LIN {X 0,Y 195.738,Z 380.154,A -85,B 0,C 180,E1 -22076.15,E2 -22076.15} C_VEL
LIN {X 0,Y 199.662,Z 372.613,A -85,B 0,C 180,E1 -22078.944,E2 -22078.944} C_VEL
LIN {X 0,Y 204.162,Z 363.072,A -85,B 0,C 180,E1 -22081.663,E2 -22081.663} C_VEL
LIN {X 0,Y 208.26,Z 353.291,A -85,B 0,C 180,E1 -22083.833,E2 -22083.833} C_VEL
LIN {X 0,Y 212.222,Z 342.404,A -85,B 0,C 180,E1 -22085.706,E2 -22085.706} C_VEL
LIN {X 0,Y 216.03,Z 330.178,A -85,B 0,C 180,E1 -22087.292,E2 -22087.292} C_VEL
LIN {X 0,Y 218.974,Z 318.329,A -85,B 0,C 180,E1 -22088.448,E2 -22088.448} C_VEL
LIN {X 0,Y 221.492,Z 304.57,A -85,B 0,C 180,E1 -22089.388,E2 -22089.388} C_VEL
LIN {X 0,Y 223.101,Z 291.496,A -85,B 0,C 180,E1 -22089.946,E2 -22089.946} C_VEL
LIN {X 0,Y 226.073,Z 252.422,A -85,B 0,C 180,E1 -22091.263,E2 -22091.263} C_VEL
LIN {X 0,Y 221.932,Z 242.001,A -85,B 0,C 180,E1 -22093.251,E2 -22093.251} C_VEL
LIN {X 0,Y 217.229,Z 232.155,A -85,B 0,C 180,E1 -22095.657,E2 -22095.657} C_VEL
LIN {X 0,Y 212.28,Z 223.234,A -85,B 0,C 180,E1 -22098.469,E2 -22098.469} C_VEL
LIN {X 0,Y 208.755,Z 217.596,A -85,B 0,C 180,E1 -22100.701,E2 -22100.701} C_VEL
LIN {X 0,Y 205.495,Z 212.523,A -85,B 0,C 180,E1 -22103.083,E2 -22103.083} C_VEL
LIN {X 0,Y 201.551,Z 206.784,A -85,B 0,C 180,E1 -22106.493,E2 -22106.493} C_VEL
LIN {X 0,Y 198.426,Z 202.606,A -85,B 0,C 180,E1 -22109.907,E2 -22109.907} C_VEL
LIN {X 0,Y 196.823,Z 200.527,A -85,B 0,C 180,E1 -22112.153,E2 -22112.153} C_VEL
LIN {X 0,Y 194.604,Z 197.984,A -85,B 0,C 180,E1 -22116.592,E2 -22116.592} C_VEL
LIN {X 0,Y 193.638,Z 197.163,A -85,B 0,C 180,E1 -22120.933,E2 -22120.933} C_VEL
LIN {X 0,Y 194.019,Z 197.379,A -85,B 0,C 180,E1 -22125.724,E2 -22125.724} C_VEL
LIN {X 0,Y 196.637,Z 198.991,A -85,B 0,C 180,E1 -22131.58,E2 -22131.58} C_VEL
LIN {X 0,Y 197.623,Z 200.557,A -85,B 0,C 180,E1 -22133.135,E2 -22133.135} C_VEL
LIN {X 0,Y 199.349,Z 203.037,A -85,B 0,C 180,E1 -22135.386,E2 -22135.386} C_VEL
LIN {X 0,Y 201.956,Z 205.11,A -85,B 0,C 180,E1 -22137.911,E2 -22137.911} C_VEL
LIN {X 0,Y 206.643,Z 212.032,A -85,B 0,C 180,E1 -22141.857,E2 -22141.857} C_VEL
LIN {X 0,Y 209.872,Z 216.687,A -85,B 0,C 180,E1 -22144.105,E2 -22144.105} C_VEL
LIN {X 0,Y 213.368,Z 222.386,A -85,B 0,C 180,E1 -22146.258,E2 -22146.258} C_VEL
LIN {X 0,Y 218.333,Z 231.127,A -85,B 0,C 180,E1 -22148.992,E2 -22148.992} C_VEL
LIN {X 0,Y 223.137,Z 241.11,A -85,B 0,C 180,E1 -22151.401,E2 -22151.401} C_VEL
LIN {X 0,Y 226.339,Z 248.713,A -85,B 0,C 180,E1 -22152.893,E2 -22152.893} C_VEL
LIN {X 0,Y 222.66,Z 293.735,A -85,B 0,C 180,E1 -22154.419,E2 -22154.419} C_VEL
LIN {X 0,Y 220.636,Z 307.167,A -85,B 0,C 180,E1 -22155.172,E2 -22155.172} C_VEL
LIN {X 0,Y 218.273,Z 318.852,A -85,B 0,C 180,E1 -22156.154,E2 -22156.154} C_VEL
LIN {X 0,Y 215.211,Z 330.433,A -85,B 0,C 180,E1 -22157.458,E2 -22157.458} C_VEL
LIN {X 0,Y 211.4,Z 342.253,A -85,B 0,C 180,E1 -22159.22,E2 -22159.22} C_VEL
LIN {X 0,Y 207.441,Z 352.476,A -85,B 0,C 180,E1 -22161.161,E2 -22161.161} C_VEL
LIN {X 0,Y 203.182,Z 362.202,A -85,B 0,C 180,E1 -22163.57,E2 -22163.57} C_VEL
LIN {X 0,Y 199.338,Z 369.905,A -85,B 0,C 180,E1 -22165.974,E2 -22165.974} C_VEL
LIN {X 0,Y 195.765,Z 376.759,A -85,B 0,C 180,E1 -22168.717,E2 -22168.717} C_VEL
LIN {X 0,Y 192.541,Z 382.26,A -85,B 0,C 180,E1 -22171.489,E2 -22171.489} C_VEL
LIN {X 0,Y 189.175,Z 387.791,A -85,B 0,C 180,E1 -22175.188,E2 -22175.188} C_VEL
LIN {X 0,Y 187.173,Z 390.817,A -85,B 0,C 180,E1 -22177.958,E2 -22177.958} C_VEL
LIN {X 0,Y 185.559,Z 393.091,A -85,B 0,C 180,E1 -22180.761,E2 -22180.761} C_VEL
LIN {X 0,Y 184.378,Z 394.674,A -85,B 0,C 180,E1 -22183.599,E2 -22183.599} C_VEL
LIN {X 0,Y 183.413,Z 395.581,A -85,B 0,C 180,E1 -22186.721,E2 -22186.721} C_VEL
LIN {X 0,Y 182.76,Z 395.654,A -85,B 0,C 180,E1 -22190.271,E2 -22190.271} C_VEL
LIN {X 0,Y 182.533,Z 394.645,A -85,B 0,C 180,E1 -22193.953,E2 -22193.953} C_VEL
LIN {X 0,Y 182.717,Z 392.379,A -85,B 0,C 180,E1 -22197.799,E2 -22197.799} C_VEL
LIN {X 0,Y 183.447,Z 388.592,A -85,B 0,C 180,E1 -22201.779,E2 -22201.779} C_VEL
LIN {X 0,Y 184.329,Z 384.06,A -85,B 0,C 180,E1 -22205.206,E2 -22205.206} C_VEL
LIN {X 0,Y 185.721,Z 377.57,A -85,B 0,C 180,E1 -22208.933,E2 -22208.933} C_VEL
LIN {X 0,Y 187.317,Z 370.754,A -85,B 0,C 180,E1 -22211.972,E2 -22211.972} C_VEL
LIN {X 0,Y 189.403,Z 362.35,A -85,B 0,C 180,E1 -22214.948,E2 -22214.948} C_VEL
LIN {X 0,Y 191.822,Z 352.236,A -85,B 0,C 180,E1 -22217.793,E2 -22217.793} C_VEL
LIN {X 0,Y 194.205,Z 341.694,A -85,B 0,C 180,E1 -22220.104,E2 -22220.104} C_VEL
LIN {X 0,Y 196.607,Z 329.365,A -85,B 0,C 180,E1 -22222.214,E2 -22222.214} C_VEL
LIN {X 0,Y 198.503,Z 317.646,A -85,B 0,C 180,E1 -22223.736,E2 -22223.736} C_VEL
LIN {X 0,Y 200.201,Z 303.923,A -85,B 0,C 180,E1 -22225.03,E2 -22225.03} C_VEL
LIN {X 0,Y 201.472,Z 291.153,A -85,B 0,C 180,E1 -22225.814,E2 -22225.814} C_VEL
LIN {X 0,Y 204.341,Z 231.553,A -85,B 0,C 180,E1 -22228.072,E2 -22228.072} C_VEL
LIN {X 0,Y 198.187,Z 214.042,A -85,B 0,C 180,E1 -22229.769,E2 -22229.769} C_VEL
LIN {X 0,Y 191.241,Z 196.738,A -85,B 0,C 180,E1 -22231.713,E2 -22231.713} C_VEL
LIN {X 0,Y 186.943,Z 189.387,A -85,B 0,C 180,E1 -22232.819,E2 -22232.819} C_VEL
LIN {X 0,Y 186.099,Z 187.307,A -85,B 0,C 180,E1 -22233.25,E2 -22233.25} C_VEL
LIN {X 0,Y 185.982,Z 186.84,A -85,B 0,C 180,E1 -22233.794,E2 -22233.794} C_VEL
LIN {X 0,Y 185.98,Z 186.809,A -85,B 0,C 180,E1 -22238.696,E2 -22238.696} C_VEL
LIN {X 0,Y 185.726,Z 186.836,A -85,B 0,C 180,E1 -22243.125,E2 -22243.125} C_VEL
LIN {X 0,Y 185.69,Z 186.842,A -85,B 0,C 180,E1 -22247.627,E2 -22247.627} C_VEL
LIN {X 0,Y 185.597,Z 186.866,A -85,B 0,C 180,E1 -22252.253,E2 -22252.253} C_VEL
LIN {X 0,Y 185.561,Z 186.846,A -85,B 0,C 180,E1 -22257.034,E2 -22257.034} C_VEL
LIN {X 0,Y 185.578,Z 186.864,A -85,B 0,C 180,E1 -22259.495,E2 -22259.495} C_VEL
LIN {X 0,Y 185.499,Z 186.853,A -85,B 0,C 180,E1 -22264.634,E2 -22264.634} C_VEL
LIN {X 0,Y 185.506,Z 186.847,A -85,B 0,C 180,E1 -22267.315,E2 -22267.315} C_VEL
LIN {X 0,Y 185.473,Z 186.879,A -85,B 0,C 180,E1 -22270.727,E2 -22270.727} C_VEL
LIN {X 0,Y 185.48,Z 186.875,A -85,B 0,C 180,E1 -22273.953,E2 -22273.953} C_VEL
LIN {X 0,Y 185.472,Z 186.839,A -85,B 0,C 180,E1 -22279.278,E2 -22279.278} C_VEL
LIN {X 0,Y 185.506,Z 186.867,A -85,B 0,C 180,E1 -22282.714,E2 -22282.714} C_VEL
LIN {X 0,Y 185.533,Z 186.866,A -85,B 0,C 180,E1 -22287.974,E2 -22287.974} C_VEL
LIN {X 0,Y 185.55,Z 186.865,A -85,B 0,C 180,E1 -22290.597,E2 -22290.597} C_VEL
LIN {X 0,Y 185.584,Z 186.862,A -85,B 0,C 180,E1 -22295.383,E2 -22295.383} C_VEL
LIN {X 0,Y 185.678,Z 186.854,A -85,B 0,C 180,E1 -22301.135,E2 -22301.135} C_VEL
LIN {X 0,Y 185.697,Z 186.839,A -85,B 0,C 180,E1 -22304.638,E2 -22304.638} C_VEL
LIN {X 0,Y 185.892,Z 186.827,A -85,B 0,C 180,E1 -22309.421,E2 -22309.421} C_VEL
LIN {X 0,Y 185.933,Z 186.815,A -85,B 0,C 180,E1 -22313.49,E2 -22313.49} C_VEL
LIN {X 0,Y 186.18,Z 186.789,A -85,B 0,C 180,E1 -22317.838,E2 -22317.838} C_VEL
LIN {X 0,Y 186.383,Z 186.749,A -85,B 0,C 180,E1 -22320.001,E2 -22320.001} C_VEL
LIN {X 0,Y 185.888,Z 186.787,A -85,B 0,C 180,E1 -22324.338,E2 -22324.338} C_VEL
LIN {X 0,Y 185.98,Z 186.816,A -85,B 0,C 180,E1 -22328.695,E2 -22328.695} C_VEL
LIN {X 0,Y 185.72,Z 186.835,A -85,B 0,C 180,E1 -22333.124,E2 -22333.124} C_VEL
LIN {X 0,Y 185.656,Z 186.834,A -85,B 0,C 180,E1 -22337.629,E2 -22337.629} C_VEL
LIN {X 0,Y 185.545,Z 186.871,A -85,B 0,C 180,E1 -22342.259,E2 -22342.259} C_VEL
LIN {X 0,Y 185.502,Z 186.856,A -85,B 0,C 180,E1 -22347.043,E2 -22347.043} C_VEL
LIN {X 0,Y 185.549,Z 186.872,A -85,B 0,C 180,E1 -22349.499,E2 -22349.499} C_VEL
LIN {X 0,Y 185.502,Z 186.86,A -85,B 0,C 180,E1 -22354.632,E2 -22354.632} C_VEL
LIN {X 0,Y 185.505,Z 186.878,A -85,B 0,C 180,E1 -22357.314,E2 -22357.314} C_VEL
LIN {X 0,Y 185.466,Z 186.869,A -85,B 0,C 180,E1 -22360.721,E2 -22360.721} C_VEL
LIN {X 0,Y 185.46,Z 186.875,A -85,B 0,C 180,E1 -22366.056,E2 -22366.056} C_VEL
LIN {X 0,Y 185.55,Z 187.033,A -85,B 0,C 180,E1 -22369.248,E2 -22369.248} C_VEL
LIN {X 0,Y 186.204,Z 189.727,A -85,B 0,C 180,E1 -22370.753,E2 -22370.753} C_VEL
LIN {X 0,Y 189.464,Z 197.093,A -85,B 0,C 180,E1 -22371.776,E2 -22371.776} C_VEL
LIN {X 0,Y 196.233,Z 213.271,A -85,B 0,C 180,E1 -22373.674,E2 -22373.674} C_VEL
LIN {X 0,Y 202.546,Z 230.72,A -85,B 0,C 180,E1 -22375.415,E2 -22375.415} C_VEL
LIN {X 0,Y 204.066,Z 243.654,A -85,B 0,C 180,E1 -22376.204,E2 -22376.204} C_VEL
LIN {X 0,Y 201.845,Z 288.233,A -85,B 0,C 180,E1 -22377.856,E2 -22377.856} C_VEL
LIN {X 0,Y 200.846,Z 294.037,A -85,B 0,C 180,E1 -22377.992,E2 -22377.992} C_VEL
LIN {X 0,Y 197.428,Z 303.347,A -85,B 0,C 180,E1 -22378.124,E2 -22378.124} C_VEL
LIN {X 0,Y 193.839,Z 312.517,A -85,B 0,C 180,E1 -22378.473,E2 -22378.473} C_VEL
LIN {X 0,Y 192.575,Z 318.098,A -85,B 0,C 180,E1 -22378.925,E2 -22378.925} C_VEL
LIN {X 0,Y 190.816,Z 329.003,A -85,B 0,C 180,E1 -22380.181,E2 -22380.181} C_VEL
LIN {X 0,Y 188.47,Z 340.49,A -85,B 0,C 180,E1 -22381.913,E2 -22381.913} C_VEL
LIN {X 0,Y 186.206,Z 351.023,A -85,B 0,C 180,E1 -22383.973,E2 -22383.973} C_VEL
LIN {X 0,Y 183.947,Z 360.69,A -85,B 0,C 180,E1 -22386.348,E2 -22386.348} C_VEL
LIN {X 0,Y 181.855,Z 369.512,A -85,B 0,C 180,E1 -22389.052,E2 -22389.052} C_VEL
LIN {X 0,Y 179.616,Z 378.019,A -85,B 0,C 180,E1 -22392.345,E2 -22392.345} C_VEL
LIN {X 0,Y 177.933,Z 384.849,A -85,B 0,C 180,E1 -22395.706,E2 -22395.706} C_VEL
LIN {X 0,Y 176.715,Z 391.092,A -85,B 0,C 180,E1 -22399.688,E2 -22399.688} C_VEL
LIN {X 0,Y 176.144,Z 395.11,A -85,B 0,C 180,E1 -22403.123,E2 -22403.123} C_VEL
LIN {X 0,Y 175.914,Z 398.454,A -85,B 0,C 180,E1 -22407.193,E2 -22407.193} C_VEL
LIN {X 0,Y 176.006,Z 399.99,A -85,B 0,C 180,E1 -22409.998,E2 -22409.998} C_VEL
LIN {X 0,Y 175.913,Z 400.846,A -85,B 0,C 180,E1 -22412.802,E2 -22412.802} C_VEL
LIN {X 0,Y 176.239,Z 401.057,A -85,B 0,C 180,E1 -22416.868,E2 -22416.868} C_VEL
LIN {X 0,Y 176.61,Z 400.64,A -85,B 0,C 180,E1 -22419.156,E2 -22419.156} C_VEL
LIN {X 0,Y 177.235,Z 399.821,A -85,B 0,C 180,E1 -22421.433,E2 -22421.433} C_VEL
LIN {X 0,Y 179.194,Z 396.958,A -85,B 0,C 180,E1 -22425.932,E2 -22425.932} C_VEL
LIN {X 0,Y 181.363,Z 393.721,A -85,B 0,C 180,E1 -22429.229,E2 -22429.229} C_VEL
LIN {X 0,Y 184.319,Z 389.441,A -85,B 0,C 180,E1 -22432.411,E2 -22432.411} C_VEL
LIN {X 0,Y 187.559,Z 384.03,A -85,B 0,C 180,E1 -22435.523,E2 -22435.523} C_VEL
LIN {X 0,Y 191.342,Z 377.304,A -85,B 0,C 180,E1 -22438.519,E2 -22438.519} C_VEL
LIN {X 0,Y 195.81,Z 369.003,A -85,B 0,C 180,E1 -22441.358,E2 -22441.358} C_VEL
LIN {X 0,Y 199.93,Z 360.528,A -85,B 0,C 180,E1 -22443.615,E2 -22443.615} C_VEL
LIN {X 0,Y 203.851,Z 351.332,A -85,B 0,C 180,E1 -22445.573,E2 -22445.573} C_VEL
LIN {X 0,Y 207.573,Z 341.406,A -85,B 0,C 180,E1 -22447.241,E2 -22447.241} C_VEL
LIN {X 0,Y 211.532,Z 328.981,A -85,B 0,C 180,E1 -22448.834,E2 -22448.834} C_VEL
LIN {X 0,Y 214.644,Z 316.652,A -85,B 0,C 180,E1 -22449.981,E2 -22449.981} C_VEL
LIN {X 0,Y 217.164,Z 302.775,A -85,B 0,C 180,E1 -22450.901,E2 -22450.901} C_VEL
LIN {X 0,Y 218.781,Z 288.708,A -85,B 0,C 180,E1 -22451.459,E2 -22451.459} C_VEL
LIN {X 0,Y 221.477,Z 254.949,A -85,B 0,C 180,E1 -22452.601,E2 -22452.601} C_VEL
LIN {X 0,Y 217.87,Z 245.778,A -85,B 0,C 180,E1 -22454.493,E2 -22454.493} C_VEL
LIN {X 0,Y 214.01,Z 237.383,A -85,B 0,C 180,E1 -22456.613,E2 -22456.613} C_VEL
LIN {X 0,Y 209.331,Z 228.687,A -85,B 0,C 180,E1 -22459.461,E2 -22459.461} C_VEL
LIN {X 0,Y 206.424,Z 223.698,A -85,B 0,C 180,E1 -22461.459,E2 -22461.459} C_VEL
LIN {X 0,Y 203.273,Z 218.661,A -85,B 0,C 180,E1 -22463.886,E2 -22463.886} C_VEL
LIN {X 0,Y 199.948,Z 213.504,A -85,B 0,C 180,E1 -22466.966,E2 -22466.966} C_VEL
LIN {X 0,Y 196.83,Z 209.093,A -85,B 0,C 180,E1 -22470.603,E2 -22470.603} C_VEL
LIN {X 0,Y 195.104,Z 206.982,A -85,B 0,C 180,E1 -22473.193,E2 -22473.193} C_VEL
LIN {X 0,Y 193.418,Z 204.91,A -85,B 0,C 180,E1 -22477.007,E2 -22477.007} C_VEL
LIN {X 0,Y 192.567,Z 204.165,A -85,B 0,C 180,E1 -22481.596,E2 -22481.596} C_VEL
LIN {X 0,Y 193.121,Z 204.542,A -85,B 0,C 180,E1 -22486.267,E2 -22486.267} C_VEL
LIN {X 0,Y 195.422,Z 205.908,A -85,B 0,C 180,E1 -22491.325,E2 -22491.325} C_VEL
LIN {X 0,Y 197.911,Z 209.845,A -85,B 0,C 180,E1 -22494.97,E2 -22494.97} C_VEL
LIN {X 0,Y 200.228,Z 211.717,A -85,B 0,C 180,E1 -22497.327,E2 -22497.327} C_VEL
LIN {X 0,Y 204.479,Z 218.281,A -85,B 0,C 180,E1 -22501.138,E2 -22501.138} C_VEL
LIN {X 0,Y 207.628,Z 223.06,A -85,B 0,C 180,E1 -22503.449,E2 -22503.449} C_VEL
LIN {X 0,Y 210.456,Z 227.855,A -85,B 0,C 180,E1 -22505.311,E2 -22505.311} C_VEL
LIN {X 0,Y 215.265,Z 236.702,A -85,B 0,C 180,E1 -22508.156,E2 -22508.156} C_VEL
LIN {X 0,Y 219.578,Z 246.025,A -85,B 0,C 180,E1 -22510.443,E2 -22510.443} C_VEL
LIN {X 0,Y 221.691,Z 251.168,A -85,B 0,C 180,E1 -22511.523,E2 -22511.523} C_VEL
LIN {X 0,Y 218.196,Z 293.227,A -85,B 0,C 180,E1 -22512.984,E2 -22512.984} C_VEL
LIN {X 0,Y 216.114,Z 306.637,A -85,B 0,C 180,E1 -22513.717,E2 -22513.717} C_VEL
LIN {X 0,Y 213.488,Z 319.191,A -85,B 0,C 180,E1 -22514.77,E2 -22514.77} C_VEL
LIN {X 0,Y 210.273,Z 330.755,A -85,B 0,C 180,E1 -22516.081,E2 -22516.081} C_VEL
LIN {X 0,Y 206.284,Z 342.543,A -85,B 0,C 180,E1 -22517.855,E2 -22517.855} C_VEL
LIN {X 0,Y 201.869,Z 353.33,A -85,B 0,C 180,E1 -22519.958,E2 -22519.958} C_VEL
LIN {X 0,Y 197.539,Z 362.643,A -85,B 0,C 180,E1 -22522.336,E2 -22522.336} C_VEL
LIN {X 0,Y 192.94,Z 371.273,A -85,B 0,C 180,E1 -22525.145,E2 -22525.145} C_VEL
LIN {X 0,Y 188.764,Z 378.65,A -85,B 0,C 180,E1 -22528.332,E2 -22528.332} C_VEL
LIN {X 0,Y 185.469,Z 383.845,A -85,B 0,C 180,E1 -22531.218,E2 -22531.218} C_VEL
LIN {X 0,Y 182.719,Z 388.005,A -85,B 0,C 180,E1 -22534.213,E2 -22534.213} C_VEL
LIN {X 0,Y 179.62,Z 392.216,A -85,B 0,C 180,E1 -22538.511,E2 -22538.511} C_VEL
LIN {X 0,Y 177.739,Z 394.503,A -85,B 0,C 180,E1 -22542.236,E2 -22542.236} C_VEL
LIN {X 0,Y 176.535,Z 395.633,A -85,B 0,C 180,E1 -22545.773,E2 -22545.773} C_VEL
LIN {X 0,Y 175.669,Z 395.73,A -85,B 0,C 180,E1 -22550.204,E2 -22550.204} C_VEL
LIN {X 0,Y 175.449,Z 394.899,A -85,B 0,C 180,E1 -22553.238,E2 -22553.238} C_VEL
LIN {X 0,Y 175.558,Z 392.775,A -85,B 0,C 180,E1 -22557.21,E2 -22557.21} C_VEL
LIN {X 0,Y 176.232,Z 389.094,A -85,B 0,C 180,E1 -22561.412,E2 -22561.412} C_VEL
LIN {X 0,Y 177.134,Z 384.659,A -85,B 0,C 180,E1 -22564.99,E2 -22564.99} C_VEL
LIN {X 0,Y 178.39,Z 378.734,A -85,B 0,C 180,E1 -22568.631,E2 -22568.631} C_VEL
LIN {X 0,Y 180.023,Z 372.156,A -85,B 0,C 180,E1 -22571.804,E2 -22571.804} C_VEL
LIN {X 0,Y 182.012,Z 364.235,A -85,B 0,C 180,E1 -22574.862,E2 -22574.862} C_VEL
LIN {X 0,Y 184.298,Z 355.24,A -85,B 0,C 180,E1 -22577.616,E2 -22577.616} C_VEL
LIN {X 0,Y 186.906,Z 344.31,A -85,B 0,C 180,E1 -22580.261,E2 -22580.261} C_VEL
LIN {X 0,Y 189.124,Z 333.821,A -85,B 0,C 180,E1 -22582.261,E2 -22582.261} C_VEL
LIN {X 0,Y 191.357,Z 321.68,A -85,B 0,C 180,E1 -22584.037,E2 -22584.037} C_VEL
LIN {X 0,Y 193.148,Z 308.919,A -85,B 0,C 180,E1 -22585.437,E2 -22585.437} C_VEL
LIN {X 0,Y 194.587,Z 295.907,A -85,B 0,C 180,E1 -22586.411,E2 -22586.411} C_VEL
LIN {X 0,Y 195.581,Z 280.594,A -85,B 0,C 180,E1 -22587.106,E2 -22587.106} C_VEL
LIN {X 0,Y 197.962,Z 233.103,A -85,B 0,C 180,E1 -22588.929,E2 -22588.929} C_VEL
LIN {X 0,Y 192.389,Z 217.271,A -85,B 0,C 180,E1 -22590.53,E2 -22590.53} C_VEL
LIN {X 0,Y 185.66,Z 200.398,A -85,B 0,C 180,E1 -22592.499,E2 -22592.499} C_VEL
LIN {X 0,Y 180.108,Z 190.85,A -85,B 0,C 180,E1 -22594.022,E2 -22594.022} C_VEL
LIN {X 0,Y 178.972,Z 188.334,A -85,B 0,C 180,E1 -22594.507,E2 -22594.507} C_VEL
LIN {X 0,Y 178.871,Z 187.736,A -85,B 0,C 180,E1 -22595.074,E2 -22595.074} C_VEL
LIN {X 0,Y 178.909,Z 187.691,A -85,B 0,C 180,E1 -22599.043,E2 -22599.043} C_VEL
LIN {X 0,Y 178.655,Z 187.718,A -85,B 0,C 180,E1 -22603.655,E2 -22603.655} C_VEL
LIN {X 0,Y 178.623,Z 187.716,A -85,B 0,C 180,E1 -22609.218,E2 -22609.218} C_VEL
LIN {X 0,Y 178.525,Z 187.727,A -85,B 0,C 180,E1 -22615.119,E2 -22615.119} C_VEL
LIN {X 0,Y 178.522,Z 187.747,A -85,B 0,C 180,E1 -22619.995,E2 -22619.995} C_VEL
LIN {X 0,Y 178.485,Z 187.729,A -85,B 0,C 180,E1 -22624.221,E2 -22624.221} C_VEL
LIN {X 0,Y 178.397,Z 187.749,A -85,B 0,C 180,E1 -22629.076,E2 -22629.076} C_VEL
LIN {X 0,Y 178.4,Z 187.762,A -85,B 0,C 180,E1 -22632.047,E2 -22632.047} C_VEL
LIN {X 0,Y 178.401,Z 187.746,A -85,B 0,C 180,E1 -22635.164,E2 -22635.164} C_VEL
LIN {X 0,Y 178.405,Z 187.715,A -85,B 0,C 180,E1 -22638.461,E2 -22638.461} C_VEL
LIN {X 0,Y 178.423,Z 187.756,A -85,B 0,C 180,E1 -22643.784,E2 -22643.784} C_VEL
LIN {X 0,Y 178.486,Z 187.75,A -85,B 0,C 180,E1 -22646.548,E2 -22646.548} C_VEL
LIN {X 0,Y 178.447,Z 187.755,A -85,B 0,C 180,E1 -22651.797,E2 -22651.797} C_VEL
LIN {X 0,Y 178.519,Z 187.742,A -85,B 0,C 180,E1 -22654.891,E2 -22654.891} C_VEL
LIN {X 0,Y 178.626,Z 187.733,A -85,B 0,C 180,E1 -22660.787,E2 -22660.787} C_VEL
LIN {X 0,Y 178.66,Z 187.722,A -85,B 0,C 180,E1 -22666.349,E2 -22666.349} C_VEL
LIN {X 0,Y 178.908,Z 187.691,A -85,B 0,C 180,E1 -22670.961,E2 -22670.961} C_VEL
LIN {X 0,Y 179.128,Z 187.668,A -85,B 0,C 180,E1 -22677.752,E2 -22677.752} C_VEL
LIN {X 0,Y 179.349,Z 187.625,A -85,B 0,C 180,E1 -22680.001,E2 -22680.001} C_VEL
LIN {X 0,Y 178.837,Z 187.665,A -85,B 0,C 180,E1 -22684.509,E2 -22684.509} C_VEL
LIN {X 0,Y 178.911,Z 187.697,A -85,B 0,C 180,E1 -22689.041,E2 -22689.041} C_VEL
LIN {X 0,Y 178.646,Z 187.711,A -85,B 0,C 180,E1 -22693.654,E2 -22693.654} C_VEL
LIN {X 0,Y 178.56,Z 187.733,A -85,B 0,C 180,E1 -22699.152,E2 -22699.152} C_VEL
LIN {X 0,Y 178.47,Z 187.728,A -85,B 0,C 180,E1 -22705.076,E2 -22705.076} C_VEL
LIN {X 0,Y 178.466,Z 187.755,A -85,B 0,C 180,E1 -22710.794,E2 -22710.794} C_VEL
LIN {X 0,Y 178.488,Z 187.731,A -85,B 0,C 180,E1 -22714.218,E2 -22714.218} C_VEL
LIN {X 0,Y 178.392,Z 187.751,A -85,B 0,C 180,E1 -22719.077,E2 -22719.077} C_VEL
LIN {X 0,Y 178.399,Z 187.76,A -85,B 0,C 180,E1 -22722.046,E2 -22722.046} C_VEL
LIN {X 0,Y 178.396,Z 187.751,A -85,B 0,C 180,E1 -22725.165,E2 -22725.165} C_VEL
LIN {X 0,Y 178.478,Z 187.975,A -85,B 0,C 180,E1 -22728.433,E2 -22728.433} C_VEL
LIN {X 0,Y 178.981,Z 189.888,A -85,B 0,C 180,E1 -22729.427,E2 -22729.427} C_VEL
LIN {X 0,Y 185.903,Z 205.264,A -85,B 0,C 180,E1 -22731.562,E2 -22731.562} C_VEL
LIN {X 0,Y 193.14,Z 223.627,A -85,B 0,C 180,E1 -22733.671,E2 -22733.671} C_VEL
LIN {X 0,Y 196.383,Z 232.984,A -85,B 0,C 180,E1 -22734.608,E2 -22734.608} C_VEL
LIN {X 0,Y 197.716,Z 244.563,A -85,B 0,C 180,E1 -22735.336,E2 -22735.336} C_VEL
LIN {X 0,Y 194.76,Z 298.7,A -85,B 0,C 180,E1 -22737.457,E2 -22737.457} C_VEL
LIN {X 0,Y 193.243,Z 312.548,A -85,B 0,C 180,E1 -22738.401,E2 -22738.401} C_VEL
LIN {X 0,Y 192.575,Z 318.098,A -85,B 0,C 180,E1 -22738.925,E2 -22738.925} C_VEL
LIN {X 0,Y 191.129,Z 323.594,A -85,B 0,C 180,E1 -22739.419,E2 -22739.419} C_VEL
LIN {X 0,Y 186.873,Z 332.206,A -85,B 0,C 180,E1 -22740.197,E2 -22740.197} C_VEL
LIN {X 0,Y 182.461,Z 340.458,A -85,B 0,C 180,E1 -22741.228,E2 -22741.228} C_VEL
LIN {X 0,Y 180.794,Z 345.385,A -85,B 0,C 180,E1 -22742.112,E2 -22742.112} C_VEL
LIN {X 0,Y 178.494,Z 355.276,A -85,B 0,C 180,E1 -22744.333,E2 -22744.333} C_VEL
LIN {X 0,Y 175.841,Z 365.552,A -85,B 0,C 180,E1 -22747.236,E2 -22747.236} C_VEL
LIN {X 0,Y 173.864,Z 373.06,A -85,B 0,C 180,E1 -22749.902,E2 -22749.902} C_VEL
LIN {X 0,Y 171.82,Z 380.848,A -85,B 0,C 180,E1 -22753.36,E2 -22753.36} C_VEL
LIN {X 0,Y 170.385,Z 387.089,A -85,B 0,C 180,E1 -22756.885,E2 -22756.885} C_VEL
LIN {X 0,Y 169.459,Z 392.013,A -85,B 0,C 180,E1 -22760.449,E2 -22760.449} C_VEL
LIN {X 0,Y 168.968,Z 395.766,A -85,B 0,C 180,E1 -22764.029,E2 -22764.029} C_VEL
LIN {X 0,Y 168.822,Z 398.459,A -85,B 0,C 180,E1 -22767.612,E2 -22767.612} C_VEL
LIN {X 0,Y 168.918,Z 399.716,A -85,B 0,C 180,E1 -22769.998,E2 -22769.998} C_VEL
LIN {X 0,Y 168.836,Z 400.584,A -85,B 0,C 180,E1 -22772.504,E2 -22772.504} C_VEL
LIN {X 0,Y 168.939,Z 400.957,A -85,B 0,C 180,E1 -22774.77,E2 -22774.77} C_VEL
LIN {X 0,Y 169.579,Z 400.602,A -85,B 0,C 180,E1 -22779.54,E2 -22779.54} C_VEL
LIN {X 0,Y 170.275,Z 399.859,A -85,B 0,C 180,E1 -22781.907,E2 -22781.907} C_VEL
LIN {X 0,Y 171.185,Z 398.703,A -85,B 0,C 180,E1 -22784.258,E2 -22784.258} C_VEL
LIN {X 0,Y 173.781,Z 395.152,A -85,B 0,C 180,E1 -22788.874,E2 -22788.874} C_VEL
LIN {X 0,Y 176.673,Z 391.337,A -85,B 0,C 180,E1 -22792.201,E2 -22792.201} C_VEL
LIN {X 0,Y 180.088,Z 386.439,A -85,B 0,C 180,E1 -22795.419,E2 -22795.419} C_VEL
LIN {X 0,Y 183.647,Z 380.584,A -85,B 0,C 180,E1 -22798.451,E2 -22798.451} C_VEL
LIN {X 0,Y 188.236,Z 372.834,A -85,B 0,C 180,E1 -22801.511,E2 -22801.511} C_VEL
LIN {X 0,Y 192.349,Z 365.182,A -85,B 0,C 180,E1 -22803.859,E2 -22803.859} C_VEL
LIN {X 0,Y 197.249,Z 354.865,A -85,B 0,C 180,E1 -22806.321,E2 -22806.321} C_VEL
LIN {X 0,Y 201.534,Z 344.461,A -85,B 0,C 180,E1 -22808.239,E2 -22808.239} C_VEL
LIN {X 0,Y 205.633,Z 332.906,A -85,B 0,C 180,E1 -22809.85,E2 -22809.85} C_VEL
LIN {X 0,Y 209.072,Z 320.831,A -85,B 0,C 180,E1 -22811.113,E2 -22811.113} C_VEL
LIN {X 0,Y 211.981,Z 307.43,A -85,B 0,C 180,E1 -22812.125,E2 -22812.125} C_VEL
LIN {X 0,Y 213.935,Z 294.223,A -85,B 0,C 180,E1 -22812.749,E2 -22812.749} C_VEL
LIN {X 0,Y 217.08,Z 257.639,A -85,B 0,C 180,E1 -22814.009,E2 -22814.009} C_VEL
LIN {X 0,Y 213.72,Z 248.932,A -85,B 0,C 180,E1 -22815.905,E2 -22815.905} C_VEL
LIN {X 0,Y 209.926,Z 240.734,A -85,B 0,C 180,E1 -22818.204,E2 -22818.204} C_VEL
LIN {X 0,Y 206.072,Z 233.369,A -85,B 0,C 180,E1 -22820.774,E2 -22820.774} C_VEL
LIN {X 0,Y 204.03,Z 229.671,A -85,B 0,C 180,E1 -22822.307,E2 -22822.307} C_VEL
LIN {X 0,Y 201.158,Z 224.843,A -85,B 0,C 180,E1 -22824.671,E2 -22824.671} C_VEL
LIN {X 0,Y 198.136,Z 220.006,A -85,B 0,C 180,E1 -22827.656,E2 -22827.656} C_VEL
LIN {X 0,Y 194.789,Z 214.896,A -85,B 0,C 180,E1 -22832.027,E2 -22832.027} C_VEL
LIN {X 0,Y 192.437,Z 211.965,A -85,B 0,C 180,E1 -22836.883,E2 -22836.883} C_VEL
LIN {X 0,Y 191.568,Z 211.136,A -85,B 0,C 180,E1 -22842.932,E2 -22842.932} C_VEL
LIN {X 0,Y 192.762,Z 212.01,A -85,B 0,C 180,E1 -22848.175,E2 -22848.175} C_VEL
LIN {X 0,Y 194.328,Z 213.048,A -85,B 0,C 180,E1 -22851.276,E2 -22851.276} C_VEL
LIN {X 0,Y 196.326,Z 216.494,A -85,B 0,C 180,E1 -22854.35,E2 -22854.35} C_VEL
LIN {X 0,Y 198.569,Z 218.425,A -85,B 0,C 180,E1 -22856.797,E2 -22856.797} C_VEL
LIN {X 0,Y 202.339,Z 224.542,A -85,B 0,C 180,E1 -22860.401,E2 -22860.401} C_VEL
LIN {X 0,Y 205.28,Z 229.162,A -85,B 0,C 180,E1 -22862.671,E2 -22862.671} C_VEL
LIN {X 0,Y 208.604,Z 235.075,A -85,B 0,C 180,E1 -22864.989,E2 -22864.989} C_VEL
LIN {X 0,Y 212.578,Z 242.955,A -85,B 0,C 180,E1 -22867.457,E2 -22867.457} C_VEL
LIN {X 0,Y 216.323,Z 251.555,A -85,B 0,C 180,E1 -22869.589,E2 -22869.589} C_VEL
LIN {X 0,Y 217.328,Z 254.041,A -85,B 0,C 180,E1 -22870.134,E2 -22870.134} C_VEL
LIN {X 0,Y 213.697,Z 294.395,A -85,B 0,C 180,E1 -22871.542,E2 -22871.542} C_VEL
LIN {X 0,Y 211.425,Z 308.144,A -85,B 0,C 180,E1 -22872.332,E2 -22872.332} C_VEL
LIN {X 0,Y 208.799,Z 319.759,A -85,B 0,C 180,E1 -22873.337,E2 -22873.337} C_VEL
LIN {X 0,Y 205.246,Z 331.776,A -85,B 0,C 180,E1 -22874.733,E2 -22874.733} C_VEL
LIN {X 0,Y 201.371,Z 342.618,A -85,B 0,C 180,E1 -22876.384,E2 -22876.384} C_VEL
LIN {X 0,Y 197.342,Z 352.222,A -85,B 0,C 180,E1 -22878.25,E2 -22878.25} C_VEL
LIN {X 0,Y 193.296,Z 360.604,A -85,B 0,C 180,E1 -22880.292,E2 -22880.292} C_VEL
LIN {X 0,Y 188.835,Z 368.898,A -85,B 0,C 180,E1 -22882.865,E2 -22882.865} C_VEL
LIN {X 0,Y 184.914,Z 375.547,A -85,B 0,C 180,E1 -22885.497,E2 -22885.497} C_VEL
LIN {X 0,Y 180.571,Z 382.214,A -85,B 0,C 180,E1 -22888.925,E2 -22888.925} C_VEL
LIN {X 0,Y 177.375,Z 386.719,A -85,B 0,C 180,E1 -22891.959,E2 -22891.959} C_VEL
LIN {X 0,Y 173.982,Z 391.206,A -85,B 0,C 180,E1 -22896.114,E2 -22896.114} C_VEL
LIN {X 0,Y 172.081,Z 393.422,A -85,B 0,C 180,E1 -22899.111,E2 -22899.111} C_VEL
LIN {X 0,Y 170.62,Z 394.961,A -85,B 0,C 180,E1 -22902.151,E2 -22902.151} C_VEL
LIN {X 0,Y 169.588,Z 395.78,A -85,B 0,C 180,E1 -22905.215,E2 -22905.215} C_VEL
LIN {X 0,Y 168.797,Z 395.942,A -85,B 0,C 180,E1 -22908.54,E2 -22908.54} C_VEL
LIN {X 0,Y 168.362,Z 395.145,A -85,B 0,C 180,E1 -22912.477,E2 -22912.477} C_VEL
LIN {X 0,Y 168.448,Z 392.791,A -85,B 0,C 180,E1 -22917.157,E2 -22917.157} C_VEL
LIN {X 0,Y 169.022,Z 389.764,A -85,B 0,C 180,E1 -22920.829,E2 -22920.829} C_VEL
LIN {X 0,Y 169.783,Z 385.969,A -85,B 0,C 180,E1 -22924.203,E2 -22924.203} C_VEL
LIN {X 0,Y 170.835,Z 381.001,A -85,B 0,C 180,E1 -22927.636,E2 -22927.636} C_VEL
LIN {X 0,Y 172.323,Z 374.923,A -85,B 0,C 180,E1 -22930.96,E2 -22930.96} C_VEL
LIN {X 0,Y 174.331,Z 367.16,A -85,B 0,C 180,E1 -22934.318,E2 -22934.318} C_VEL
LIN {X 0,Y 176.704,Z 358.242,A -85,B 0,C 180,E1 -22937.367,E2 -22937.367} C_VEL
LIN {X 0,Y 179.185,Z 348.418,A -85,B 0,C 180,E1 -22940.04,E2 -22940.04} C_VEL
LIN {X 0,Y 181.591,Z 338.292,A -85,B 0,C 180,E1 -22942.217,E2 -22942.217} C_VEL
LIN {X 0,Y 183.95,Z 326.454,A -85,B 0,C 180,E1 -22944.203,E2 -22944.203} C_VEL
LIN {X 0,Y 185.98,Z 313.89,A -85,B 0,C 180,E1 -22945.804,E2 -22945.804} C_VEL
LIN {X 0,Y 187.698,Z 300.563,A -85,B 0,C 180,E1 -22946.984,E2 -22946.984} C_VEL
LIN {X 0,Y 188.84,Z 287.291,A -85,B 0,C 180,E1 -22947.736,E2 -22947.736} C_VEL
LIN {X 0,Y 191.604,Z 234.703,A -85,B 0,C 180,E1 -22949.82,E2 -22949.82} C_VEL
LIN {X 0,Y 186.211,Z 219.316,A -85,B 0,C 180,E1 -22951.464,E2 -22951.464} C_VEL
LIN {X 0,Y 180.269,Z 204.24,A -85,B 0,C 180,E1 -22953.294,E2 -22953.294} C_VEL
LIN {X 0,Y 172.183,Z 190.005,A -85,B 0,C 180,E1 -22955.713,E2 -22955.713} C_VEL
LIN {X 0,Y 171.865,Z 188.799,A -85,B 0,C 180,E1 -22956.165,E2 -22956.165} C_VEL
LIN {X 0,Y 171.846,Z 188.573,A -85,B 0,C 180,E1 -22959.418,E2 -22959.418} C_VEL
LIN {X 0,Y 171.573,Z 188.604,A -85,B 0,C 180,E1 -22964.23,E2 -22964.23} C_VEL
LIN {X 0,Y 171.544,Z 188.598,A -85,B 0,C 180,E1 -22969.564,E2 -22969.564} C_VEL
LIN {X 0,Y 171.462,Z 188.602,A -85,B 0,C 180,E1 -22975.613,E2 -22975.613} C_VEL
LIN {X 0,Y 171.44,Z 188.63,A -85,B 0,C 180,E1 -22980.588,E2 -22980.588} C_VEL
LIN {X 0,Y 171.393,Z 188.602,A -85,B 0,C 180,E1 -22985.037,E2 -22985.037} C_VEL
LIN {X 0,Y 171.359,Z 188.623,A -85,B 0,C 180,E1 -22988.809,E2 -22988.809} C_VEL
LIN {X 0,Y 171.328,Z 188.633,A -85,B 0,C 180,E1 -22994.218,E2 -22994.218} C_VEL
LIN {X 0,Y 171.337,Z 188.594,A -85,B 0,C 180,E1 -22998.983,E2 -22998.983} C_VEL
LIN {X 0,Y 171.387,Z 188.62,A -85,B 0,C 180,E1 -23002.042,E2 -23002.042} C_VEL
LIN {X 0,Y 171.4,Z 188.634,A -85,B 0,C 180,E1 -23005.095,E2 -23005.095} C_VEL
LIN {X 0,Y 171.411,Z 188.624,A -85,B 0,C 180,E1 -23010.529,E2 -23010.529} C_VEL
LIN {X 0,Y 171.445,Z 188.618,A -85,B 0,C 180,E1 -23015.801,E2 -23015.801} C_VEL
LIN {X 0,Y 171.582,Z 188.61,A -85,B 0,C 180,E1 -23020.873,E2 -23020.873} C_VEL
LIN {X 0,Y 171.578,Z 188.6,A -85,B 0,C 180,E1 -23025.774,E2 -23025.774} C_VEL
LIN {X 0,Y 171.847,Z 188.571,A -85,B 0,C 180,E1 -23030.586,E2 -23030.586} C_VEL
LIN {X 0,Y 171.786,Z 188.585,A -85,B 0,C 180,E1 -23035.308,E2 -23035.308} C_VEL
LIN {X 0,Y 172.313,Z 188.5,A -85,B 0,C 180,E1 -23040.001,E2 -23040.001} C_VEL
LIN {X 0,Y 171.787,Z 188.542,A -85,B 0,C 180,E1 -23044.694,E2 -23044.694} C_VEL
LIN {X 0,Y 171.849,Z 188.578,A -85,B 0,C 180,E1 -23049.416,E2 -23049.416} C_VEL
LIN {X 0,Y 171.56,Z 188.584,A -85,B 0,C 180,E1 -23054.23,E2 -23054.23} C_VEL
LIN {X 0,Y 171.484,Z 188.617,A -85,B 0,C 180,E1 -23059.499,E2 -23059.499} C_VEL
LIN {X 0,Y 171.408,Z 188.605,A -85,B 0,C 180,E1 -23065.569,E2 -23065.569} C_VEL
LIN {X 0,Y 171.423,Z 188.633,A -85,B 0,C 180,E1 -23070.572,E2 -23070.572} C_VEL
LIN {X 0,Y 171.398,Z 188.618,A -85,B 0,C 180,E1 -23075.035,E2 -23075.035} C_VEL
LIN {X 0,Y 171.348,Z 188.63,A -85,B 0,C 180,E1 -23078.801,E2 -23078.801} C_VEL
LIN {X 0,Y 171.324,Z 188.634,A -85,B 0,C 180,E1 -23084.218,E2 -23084.218} C_VEL
LIN {X 0,Y 171.398,Z 188.882,A -85,B 0,C 180,E1 -23087.493,E2 -23087.493} C_VEL
LIN {X 0,Y 171.722,Z 190.075,A -85,B 0,C 180,E1 -23087.958,E2 -23087.958} C_VEL
LIN {X 0,Y 177.228,Z 201.676,A -85,B 0,C 180,E1 -23089.766,E2 -23089.766} C_VEL
LIN {X 0,Y 183.856,Z 217.381,A -85,B 0,C 180,E1 -23091.809,E2 -23091.809} C_VEL
LIN {X 0,Y 190.215,Z 235.132,A -85,B 0,C 180,E1 -23093.758,E2 -23093.758} C_VEL
LIN {X 0,Y 191.343,Z 245.132,A -85,B 0,C 180,E1 -23094.414,E2 -23094.414} C_VEL
LIN {X 0,Y 188.38,Z 297.877,A -85,B 0,C 180,E1 -23096.531,E2 -23096.531} C_VEL
LIN {X 0,Y 186.879,Z 311.186,A -85,B 0,C 180,E1 -23097.433,E2 -23097.433} C_VEL
LIN {X 0,Y 185.125,Z 323.563,A -85,B 0,C 180,E1 -23098.691,E2 -23098.691} C_VEL
LIN {X 0,Y 182.899,Z 335.508,A -85,B 0,C 180,E1 -23100.346,E2 -23100.346} C_VEL
LIN {X 0,Y 180.794,Z 345.385,A -85,B 0,C 180,E1 -23102.112,E2 -23102.112} C_VEL
LIN {X 0,Y 179.123,Z 350.246,A -85,B 0,C 180,E1 -23103.078,E2 -23103.078} C_VEL
LIN {X 0,Y 174.573,Z 357.675,A -85,B 0,C 180,E1 -23104.627,E2 -23104.627} C_VEL
LIN {X 0,Y 169.964,Z 364.577,A -85,B 0,C 180,E1 -23106.422,E2 -23106.422} C_VEL
LIN {X 0,Y 168.235,Z 368.59,A -85,B 0,C 180,E1 -23107.746,E2 -23107.746} C_VEL
LIN {X 0,Y 166.079,Z 376.314,A -85,B 0,C 180,E1 -23110.853,E2 -23110.853} C_VEL
LIN {X 0,Y 164.118,Z 383.436,A -85,B 0,C 180,E1 -23114.474,E2 -23114.474} C_VEL
LIN {X 0,Y 162.723,Z 389.938,A -85,B 0,C 180,E1 -23118.791,E2 -23118.791} C_VEL
LIN {X 0,Y 162.025,Z 394.174,A -85,B 0,C 180,E1 -23122.521,E2 -23122.521} C_VEL
LIN {X 0,Y 161.8,Z 396.401,A -85,B 0,C 180,E1 -23125.014,E2 -23125.014} C_VEL
LIN {X 0,Y 161.739,Z 398.453,A -85,B 0,C 180,E1 -23128.068,E2 -23128.068} C_VEL
LIN {X 0,Y 161.824,Z 399.43,A -85,B 0,C 180,E1 -23129.997,E2 -23129.997} C_VEL
LIN {X 0,Y 161.76,Z 400.322,A -85,B 0,C 180,E1 -23132.487,E2 -23132.487} C_VEL
LIN {X 0,Y 161.859,Z 400.815,A -85,B 0,C 180,E1 -23134.979,E2 -23134.979} C_VEL
LIN {X 0,Y 162.13,Z 400.882,A -85,B 0,C 180,E1 -23137.469,E2 -23137.469} C_VEL
LIN {X 0,Y 163.305,Z 399.874,A -85,B 0,C 180,E1 -23142.423,E2 -23142.423} C_VEL
LIN {X 0,Y 164.3,Z 398.802,A -85,B 0,C 180,E1 -23144.869,E2 -23144.869} C_VEL
LIN {X 0,Y 165.527,Z 397.301,A -85,B 0,C 180,E1 -23147.287,E2 -23147.287} C_VEL
LIN {X 0,Y 168.039,Z 394.295,A -85,B 0,C 180,E1 -23150.821,E2 -23150.821} C_VEL
LIN {X 0,Y 171.333,Z 390.266,A -85,B 0,C 180,E1 -23154.214,E2 -23154.214} C_VEL
LIN {X 0,Y 175.212,Z 384.552,A -85,B 0,C 180,E1 -23157.86,E2 -23157.86} C_VEL
LIN {X 0,Y 179.887,Z 377.525,A -85,B 0,C 180,E1 -23161.172,E2 -23161.172} C_VEL
LIN {X 0,Y 184.8,Z 369.349,A -85,B 0,C 180,E1 -23164.118,E2 -23164.118} C_VEL
LIN {X 0,Y 189.312,Z 361.041,A -85,B 0,C 180,E1 -23166.437,E2 -23166.437} C_VEL
LIN {X 0,Y 194.147,Z 350.895,A -85,B 0,C 180,E1 -23168.637,E2 -23168.637} C_VEL
LIN {X 0,Y 198.234,Z 340.969,A -85,B 0,C 180,E1 -23170.314,E2 -23170.314} C_VEL
LIN {X 0,Y 201.964,Z 330.263,A -85,B 0,C 180,E1 -23171.718,E2 -23171.718} C_VEL
LIN {X 0,Y 205.596,Z 317.445,A -85,B 0,C 180,E1 -23172.96,E2 -23172.96} C_VEL
LIN {X 0,Y 208.306,Z 304.179,A -85,B 0,C 180,E1 -23173.863,E2 -23173.863} C_VEL
LIN {X 0,Y 210.099,Z 291.231,A -85,B 0,C 180,E1 -23174.413,E2 -23174.413} C_VEL
LIN {X 0,Y 212.747,Z 260.131,A -85,B 0,C 180,E1 -23175.516,E2 -23175.516} C_VEL
LIN {X 0,Y 209.715,Z 252.086,A -85,B 0,C 180,E1 -23177.422,E2 -23177.422} C_VEL
LIN {X 0,Y 205.94,Z 243.883,A -85,B 0,C 180,E1 -23179.913,E2 -23179.913} C_VEL
LIN {X 0,Y 202.202,Z 236.463,A -85,B 0,C 180,E1 -23182.764,E2 -23182.764} C_VEL
LIN {X 0,Y 198.988,Z 230.882,A -85,B 0,C 180,E1 -23185.59,E2 -23185.59} C_VEL
LIN {X 0,Y 196.359,Z 226.489,A -85,B 0,C 180,E1 -23188.355,E2 -23188.355} C_VEL
LIN {X 0,Y 193.322,Z 221.573,A -85,B 0,C 180,E1 -23192.644,E2 -23192.644} C_VEL
LIN {X 0,Y 191.253,Z 218.899,A -85,B 0,C 180,E1 -23197.303,E2 -23197.303} C_VEL
LIN {X 0,Y 190.537,Z 218.16,A -85,B 0,C 180,E1 -23202.837,E2 -23202.837} C_VEL
LIN {X 0,Y 191.988,Z 219.167,A -85,B 0,C 180,E1 -23208.763,E2 -23208.763} C_VEL
LIN {X 0,Y 193.071,Z 219.95,A -85,B 0,C 180,E1 -23210.913,E2 -23210.913} C_VEL
LIN {X 0,Y 194.811,Z 223.173,A -85,B 0,C 180,E1 -23213.786,E2 -23213.786} C_VEL
LIN {X 0,Y 196.892,Z 225.092,A -85,B 0,C 180,E1 -23216.226,E2 -23216.226} C_VEL
LIN {X 0,Y 200.275,Z 230.811,A -85,B 0,C 180,E1 -23219.65,E2 -23219.65} C_VEL
LIN {X 0,Y 203.282,Z 235.796,A -85,B 0,C 180,E1 -23222.118,E2 -23222.118} C_VEL
LIN {X 0,Y 206.557,Z 242.131,A -85,B 0,C 180,E1 -23224.546,E2 -23224.546} C_VEL
LIN {X 0,Y 209.962,Z 249.254,A -85,B 0,C 180,E1 -23226.761,E2 -23226.761} C_VEL
LIN {X 0,Y 213.029,Z 256.828,A -85,B 0,C 180,E1 -23228.656,E2 -23228.656} C_VEL
LIN {X 0,Y 209.568,Z 294.193,A -85,B 0,C 180,E1 -23229.976,E2 -23229.976} C_VEL
LIN {X 0,Y 207.143,Z 308.273,A -85,B 0,C 180,E1 -23230.77,E2 -23230.77} C_VEL
LIN {X 0,Y 203.985,Z 321.382,A -85,B 0,C 180,E1 -23231.929,E2 -23231.929} C_VEL
LIN {X 0,Y 199.993,Z 334.003,A -85,B 0,C 180,E1 -23233.453,E2 -23233.453} C_VEL
LIN {X 0,Y 195.745,Z 344.975,A -85,B 0,C 180,E1 -23235.235,E2 -23235.235} C_VEL
LIN {X 0,Y 190.682,Z 355.828,A -85,B 0,C 180,E1 -23237.518,E2 -23237.518} C_VEL
LIN {X 0,Y 186.144,Z 364.389,A -85,B 0,C 180,E1 -23239.864,E2 -23239.864} C_VEL
LIN {X 0,Y 181.014,Z 372.862,A -85,B 0,C 180,E1 -23242.845,E2 -23242.845} C_VEL
LIN {X 0,Y 176.689,Z 379.487,A -85,B 0,C 180,E1 -23245.946,E2 -23245.946} C_VEL
LIN {X 0,Y 172.72,Z 384.894,A -85,B 0,C 180,E1 -23249.226,E2 -23249.226} C_VEL
LIN {X 0,Y 169.441,Z 389.083,A -85,B 0,C 180,E1 -23252.628,E2 -23252.628} C_VEL
LIN {X 0,Y 166.383,Z 392.592,A -85,B 0,C 180,E1 -23256.63,E2 -23256.63} C_VEL
LIN {X 0,Y 164.495,Z 394.477,A -85,B 0,C 180,E1 -23259.855,E2 -23259.855} C_VEL
LIN {X 0,Y 162.924,Z 395.754,A -85,B 0,C 180,E1 -23263.643,E2 -23263.643} C_VEL
LIN {X 0,Y 161.884,Z 396.084,A -85,B 0,C 180,E1 -23267.563,E2 -23267.563} C_VEL
LIN {X 0,Y 161.28,Z 395.128,A -85,B 0,C 180,E1 -23272.409,E2 -23272.409} C_VEL
LIN {X 0,Y 161.255,Z 393.504,A -85,B 0,C 180,E1 -23275.9,E2 -23275.9} C_VEL
LIN {X 0,Y 161.832,Z 390.28,A -85,B 0,C 180,E1 -23280.289,E2 -23280.289} C_VEL
LIN {X 0,Y 162.718,Z 385.919,A -85,B 0,C 180,E1 -23284.414,E2 -23284.414} C_VEL
LIN {X 0,Y 164.05,Z 379.843,A -85,B 0,C 180,E1 -23288.649,E2 -23288.649} C_VEL
LIN {X 0,Y 165.731,Z 373.456,A -85,B 0,C 180,E1 -23292.098,E2 -23292.098} C_VEL
LIN {X 0,Y 167.807,Z 365.668,A -85,B 0,C 180,E1 -23295.449,E2 -23295.449} C_VEL
LIN {X 0,Y 170.365,Z 356.632,A -85,B 0,C 180,E1 -23298.528,E2 -23298.528} C_VEL
LIN {X 0,Y 172.976,Z 346.519,A -85,B 0,C 180,E1 -23301.239,E2 -23301.239} C_VEL
LIN {X 0,Y 175.419,Z 336.057,A -85,B 0,C 180,E1 -23303.455,E2 -23303.455} C_VEL
LIN {X 0,Y 177.934,Z 323.764,A -85,B 0,C 180,E1 -23305.472,E2 -23305.472} C_VEL
LIN {X 0,Y 179.994,Z 310.539,A -85,B 0,C 180,E1 -23307.065,E2 -23307.065} C_VEL
LIN {X 0,Y 181.614,Z 297.442,A -85,B 0,C 180,E1 -23308.155,E2 -23308.155} C_VEL
LIN {X 0,Y 182.717,Z 282.748,A -85,B 0,C 180,E1 -23308.89,E2 -23308.89} C_VEL
LIN {X 0,Y 185.323,Z 236.437,A -85,B 0,C 180,E1 -23310.761,E2 -23310.761} C_VEL
LIN {X 0,Y 180.519,Z 222.607,A -85,B 0,C 180,E1 -23312.301,E2 -23312.301} C_VEL
LIN {X 0,Y 174.781,Z 207.881,A -85,B 0,C 180,E1 -23314.169,E2 -23314.169} C_VEL
LIN {X 0,Y 165.976,Z 192.552,A -85,B 0,C 180,E1 -23316.897,E2 -23316.897} C_VEL
LIN {X 0,Y 164.923,Z 190.096,A -85,B 0,C 180,E1 -23317.424,E2 -23317.424} C_VEL
LIN {X 0,Y 164.81,Z 189.495,A -85,B 0,C 180,E1 -23317.969,E2 -23317.969} C_VEL
LIN {X 0,Y 164.594,Z 189.467,A -85,B 0,C 180,E1 -23322.33,E2 -23322.33} C_VEL
LIN {X 0,Y 164.482,Z 189.482,A -85,B 0,C 180,E1 -23327.406,E2 -23327.406} C_VEL
LIN {X 0,Y 164.473,Z 189.48,A -85,B 0,C 180,E1 -23329.992,E2 -23329.992} C_VEL
LIN {X 0,Y 164.388,Z 189.48,A -85,B 0,C 180,E1 -23336.132,E2 -23336.132} C_VEL
LIN {X 0,Y 164.374,Z 189.511,A -85,B 0,C 180,E1 -23341.229,E2 -23341.229} C_VEL
LIN {X 0,Y 164.295,Z 189.481,A -85,B 0,C 180,E1 -23346.792,E2 -23346.792} C_VEL
LIN {X 0,Y 164.292,Z 189.512,A -85,B 0,C 180,E1 -23349.918,E2 -23349.918} C_VEL
LIN {X 0,Y 164.281,Z 189.517,A -85,B 0,C 180,E1 -23353.344,E2 -23353.344} C_VEL
LIN {X 0,Y 164.295,Z 189.477,A -85,B 0,C 180,E1 -23356.811,E2 -23356.811} C_VEL
LIN {X 0,Y 164.297,Z 189.479,A -85,B 0,C 180,E1 -23360.354,E2 -23360.354} C_VEL
LIN {X 0,Y 164.332,Z 189.513,A -85,B 0,C 180,E1 -23364.351,E2 -23364.351} C_VEL
LIN {X 0,Y 164.373,Z 189.495,A -85,B 0,C 180,E1 -23369.132,E2 -23369.132} C_VEL
LIN {X 0,Y 164.398,Z 189.501,A -85,B 0,C 180,E1 -23374.692,E2 -23374.692} C_VEL
LIN {X 0,Y 164.489,Z 189.493,A -85,B 0,C 180,E1 -23380.053,E2 -23380.053} C_VEL
LIN {X 0,Y 164.508,Z 189.477,A -85,B 0,C 180,E1 -23385.149,E2 -23385.149} C_VEL
LIN {X 0,Y 164.768,Z 189.454,A -85,B 0,C 180,E1 -23390.178,E2 -23390.178} C_VEL
LIN {X 0,Y 164.823,Z 189.439,A -85,B 0,C 180,E1 -23392.652,E2 -23392.652} C_VEL
LIN {X 0,Y 165.278,Z 189.374,A -85,B 0,C 180,E1 -23400.001,E2 -23400.001} C_VEL
LIN {X 0,Y 164.826,Z 189.441,A -85,B 0,C 180,E1 -23407.35,E2 -23407.35} C_VEL
LIN {X 0,Y 164.707,Z 189.467,A -85,B 0,C 180,E1 -23411.059,E2 -23411.059} C_VEL
LIN {X 0,Y 164.44,Z 189.468,A -85,B 0,C 180,E1 -23417.409,E2 -23417.409} C_VEL
LIN {X 0,Y 164.425,Z 189.5,A -85,B 0,C 180,E1 -23419.996,E2 -23419.996} C_VEL
LIN {X 0,Y 164.344,Z 189.483,A -85,B 0,C 180,E1 -23426.094,E2 -23426.094} C_VEL
LIN {X 0,Y 164.359,Z 189.509,A -85,B 0,C 180,E1 -23431.214,E2 -23431.214} C_VEL
LIN {X 0,Y 164.285,Z 189.521,A -85,B 0,C 180,E1 -23436.793,E2 -23436.793} C_VEL
LIN {X 0,Y 164.291,Z 189.503,A -85,B 0,C 180,E1 -23439.918,E2 -23439.918} C_VEL
LIN {X 0,Y 164.307,Z 189.595,A -85,B 0,C 180,E1 -23445.764,E2 -23445.764} C_VEL
LIN {X 0,Y 164.426,Z 190.308,A -85,B 0,C 180,E1 -23446.272,E2 -23446.272} C_VEL
LIN {X 0,Y 165.982,Z 193.33,A -85,B 0,C 180,E1 -23446.921,E2 -23446.921} C_VEL
LIN {X 0,Y 170.539,Z 202.546,A -85,B 0,C 180,E1 -23448.442,E2 -23448.442} C_VEL
LIN {X 0,Y 177.808,Z 219.724,A -85,B 0,C 180,E1 -23450.83,E2 -23450.83} C_VEL
LIN {X 0,Y 184.104,Z 237.475,A -85,B 0,C 180,E1 -23452.863,E2 -23452.863} C_VEL
LIN {X 0,Y 185,Z 246.253,A -85,B 0,C 180,E1 -23453.452,E2 -23453.452} C_VEL
LIN {X 0,Y 181.969,Z 298.136,A -85,B 0,C 180,E1 -23455.606,E2 -23455.606} C_VEL
LIN {X 0,Y 180.306,Z 312.048,A -85,B 0,C 180,E1 -23456.592,E2 -23456.592} C_VEL
LIN {X 0,Y 178.516,Z 324.16,A -85,B 0,C 180,E1 -23457.892,E2 -23457.892} C_VEL
LIN {X 0,Y 176.07,Z 336.723,A -85,B 0,C 180,E1 -23459.737,E2 -23459.737} C_VEL
LIN {X 0,Y 173.8,Z 346.689,A -85,B 0,C 180,E1 -23461.629,E2 -23461.629} C_VEL
LIN {X 0,Y 171.126,Z 357.457,A -85,B 0,C 180,E1 -23464.224,E2 -23464.224} C_VEL
LIN {X 0,Y 168.829,Z 366.139,A -85,B 0,C 180,E1 -23466.876,E2 -23466.876} C_VEL
LIN {X 0,Y 168.235,Z 368.59,A -85,B 0,C 180,E1 -23467.746,E2 -23467.746} C_VEL
LIN {X 0,Y 166.541,Z 372.48,A -85,B 0,C 180,E1 -23469.154,E2 -23469.154} C_VEL
LIN {X 0,Y 162.083,Z 378.236,A -85,B 0,C 180,E1 -23471.508,E2 -23471.508} C_VEL
LIN {X 0,Y 157.79,Z 383.318,A -85,B 0,C 180,E1 -23474.158,E2 -23474.158} C_VEL
LIN {X 0,Y 156.405,Z 386.152,A -85,B 0,C 180,E1 -23475.987,E2 -23475.987} C_VEL
LIN {X 0,Y 155.431,Z 390.903,A -85,B 0,C 180,E1 -23479.577,E2 -23479.577} C_VEL
LIN {X 0,Y 154.847,Z 394.879,A -85,B 0,C 180,E1 -23483.482,E2 -23483.482} C_VEL
LIN {X 0,Y 154.655,Z 398.543,A -85,B 0,C 180,E1 -23488.764,E2 -23488.764} C_VEL
LIN {X 0,Y 154.668,Z 400.081,A -85,B 0,C 180,E1 -23492.602,E2 -23492.602} C_VEL
LIN {X 0,Y 154.791,Z 400.637,A -85,B 0,C 180,E1 -23495.207,E2 -23495.207} C_VEL
LIN {X 0,Y 155.066,Z 400.793,A -85,B 0,C 180,E1 -23497.812,E2 -23497.812} C_VEL
LIN {X 0,Y 156.361,Z 399.894,A -85,B 0,C 180,E1 -23502.984,E2 -23502.984} C_VEL
LIN {X 0,Y 158.737,Z 397.486,A -85,B 0,C 180,E1 -23508.051,E2 -23508.051} C_VEL
LIN {X 0,Y 161.436,Z 394.574,A -85,B 0,C 180,E1 -23511.715,E2 -23511.715} C_VEL
LIN {X 0,Y 164.894,Z 390.66,A -85,B 0,C 180,E1 -23515.224,E2 -23515.224} C_VEL
LIN {X 0,Y 168.795,Z 385.388,A -85,B 0,C 180,E1 -23518.828,E2 -23518.828} C_VEL
LIN {X 0,Y 173.903,Z 378.287,A -85,B 0,C 180,E1 -23522.373,E2 -23522.373} C_VEL
LIN {X 0,Y 179.028,Z 370.334,A -85,B 0,C 180,E1 -23525.379,E2 -23525.379} C_VEL
LIN {X 0,Y 184.685,Z 360.487,A -85,B 0,C 180,E1 -23528.194,E2 -23528.194} C_VEL
LIN {X 0,Y 189.781,Z 350.228,A -85,B 0,C 180,E1 -23530.392,E2 -23530.392} C_VEL
LIN {X 0,Y 194.067,Z 340.178,A -85,B 0,C 180,E1 -23532.061,E2 -23532.061} C_VEL
LIN {X 0,Y 197.966,Z 329.308,A -85,B 0,C 180,E1 -23533.455,E2 -23533.455} C_VEL
LIN {X 0,Y 201.328,Z 317.846,A -85,B 0,C 180,E1 -23534.554,E2 -23534.554} C_VEL
LIN {X 0,Y 204.228,Z 304.423,A -85,B 0,C 180,E1 -23535.474,E2 -23535.474} C_VEL
LIN {X 0,Y 206.194,Z 290.858,A -85,B 0,C 180,E1 -23536.05,E2 -23536.05} C_VEL
LIN {X 0,Y 208.685,Z 262.832,A -85,B 0,C 180,E1 -23537.064,E2 -23537.064} C_VEL
LIN {X 0,Y 205.438,Z 254.361,A -85,B 0,C 180,E1 -23539.289,E2 -23539.289} C_VEL
LIN {X 0,Y 201.876,Z 246.461,A -85,B 0,C 180,E1 -23541.986,E2 -23541.986} C_VEL
LIN {X 0,Y 199.187,Z 241.279,A -85,B 0,C 180,E1 -23544.24,E2 -23544.24} C_VEL
LIN {X 0,Y 196.992,Z 237.09,A -85,B 0,C 180,E1 -23546.407,E2 -23546.407} C_VEL
LIN {X 0,Y 194.782,Z 233.153,A -85,B 0,C 180,E1 -23548.907,E2 -23548.907} C_VEL
LIN {X 0,Y 192.029,Z 228.408,A -85,B 0,C 180,E1 -23553.028,E2 -23553.028} C_VEL
LIN {X 0,Y 190.149,Z 225.874,A -85,B 0,C 180,E1 -23557.512,E2 -23557.512} C_VEL
LIN {X 0,Y 189.501,Z 225.191,A -85,B 0,C 180,E1 -23562.74,E2 -23562.74} C_VEL
LIN {X 0,Y 190.701,Z 226.083,A -85,B 0,C 180,E1 -23568.199,E2 -23568.199} C_VEL
LIN {X 0,Y 191.756,Z 226.771,A -85,B 0,C 180,E1 -23570.415,E2 -23570.415} C_VEL
LIN {X 0,Y 193.337,Z 229.871,A -85,B 0,C 180,E1 -23573.243,E2 -23573.243} C_VEL
LIN {X 0,Y 195.285,Z 231.817,A -85,B 0,C 180,E1 -23575.68,E2 -23575.68} C_VEL
LIN {X 0,Y 198.182,Z 236.909,A -85,B 0,C 180,E1 -23578.795,E2 -23578.795} C_VEL
LIN {X 0,Y 201.103,Z 242.133,A -85,B 0,C 180,E1 -23581.401,E2 -23581.401} C_VEL
LIN {X 0,Y 204.468,Z 249,A -85,B 0,C 180,E1 -23584.028,E2 -23584.028} C_VEL
LIN {X 0,Y 207.733,Z 256.445,A -85,B 0,C 180,E1 -23586.286,E2 -23586.286} C_VEL
LIN {X 0,Y 209.009,Z 259.773,A -85,B 0,C 180,E1 -23587.134,E2 -23587.134} C_VEL
LIN {X 0,Y 205.596,Z 294.386,A -85,B 0,C 180,E1 -23588.357,E2 -23588.357} C_VEL
LIN {X 0,Y 203.269,Z 307.416,A -85,B 0,C 180,E1 -23589.077,E2 -23589.077} C_VEL
LIN {X 0,Y 200.362,Z 319.496,A -85,B 0,C 180,E1 -23590.1,E2 -23590.1} C_VEL
LIN {X 0,Y 196.351,Z 332.031,A -85,B 0,C 180,E1 -23591.541,E2 -23591.541} C_VEL
LIN {X 0,Y 192.163,Z 342.719,A -85,B 0,C 180,E1 -23593.168,E2 -23593.168} C_VEL
LIN {X 0,Y 187.425,Z 353.034,A -85,B 0,C 180,E1 -23595.216,E2 -23595.216} C_VEL
LIN {X 0,Y 182.361,Z 362.316,A -85,B 0,C 180,E1 -23597.59,E2 -23597.59} C_VEL
LIN {X 0,Y 177.278,Z 370.576,A -85,B 0,C 180,E1 -23600.341,E2 -23600.341} C_VEL
LIN {X 0,Y 172.725,Z 377.264,A -85,B 0,C 180,E1 -23603.235,E2 -23603.235} C_VEL
LIN {X 0,Y 168.622,Z 382.773,A -85,B 0,C 180,E1 -23606.311,E2 -23606.311} C_VEL
LIN {X 0,Y 163.668,Z 388.714,A -85,B 0,C 180,E1 -23610.823,E2 -23610.823} C_VEL
LIN {X 0,Y 160.427,Z 392.203,A -85,B 0,C 180,E1 -23614.714,E2 -23614.714} C_VEL
LIN {X 0,Y 157.989,Z 394.48,A -85,B 0,C 180,E1 -23618.518,E2 -23618.518} C_VEL
LIN {X 0,Y 155.729,Z 396.052,A -85,B 0,C 180,E1 -23623.779,E2 -23623.779} C_VEL
LIN {X 0,Y 154.875,Z 396.182,A -85,B 0,C 180,E1 -23627.108,E2 -23627.108} C_VEL
LIN {X 0,Y 154.277,Z 395.614,A -85,B 0,C 180,E1 -23630.751,E2 -23630.751} C_VEL
LIN {X 0,Y 154.134,Z 393.853,A -85,B 0,C 180,E1 -23635.157,E2 -23635.157} C_VEL
LIN {X 0,Y 154.661,Z 390.515,A -85,B 0,C 180,E1 -23640.013,E2 -23640.013} C_VEL
LIN {X 0,Y 155.63,Z 385.917,A -85,B 0,C 180,E1 -23644.575,E2 -23644.575} C_VEL
LIN {X 0,Y 156.789,Z 380.897,A -85,B 0,C 180,E1 -23648.3,E2 -23648.3} C_VEL
LIN {X 0,Y 158.804,Z 373.312,A -85,B 0,C 180,E1 -23652.622,E2 -23652.622} C_VEL
LIN {X 0,Y 160.978,Z 365.472,A -85,B 0,C 180,E1 -23656.109,E2 -23656.109} C_VEL
LIN {X 0,Y 163.792,Z 355.862,A -85,B 0,C 180,E1 -23659.456,E2 -23659.456} C_VEL
LIN {X 0,Y 166.736,Z 344.828,A -85,B 0,C 180,E1 -23662.434,E2 -23662.434} C_VEL
LIN {X 0,Y 169.369,Z 333.614,A -85,B 0,C 180,E1 -23664.786,E2 -23664.786} C_VEL
LIN {X 0,Y 171.947,Z 320.951,A -85,B 0,C 180,E1 -23666.781,E2 -23666.781} C_VEL
LIN {X 0,Y 173.895,Z 308.128,A -85,B 0,C 180,E1 -23668.286,E2 -23668.286} C_VEL
LIN {X 0,Y 175.541,Z 294.353,A -85,B 0,C 180,E1 -23669.343,E2 -23669.343} C_VEL
LIN {X 0,Y 177.12,Z 270.589,A -85,B 0,C 180,E1 -23670.413,E2 -23670.413} C_VEL
LIN {X 0,Y 178.993,Z 237.943,A -85,B 0,C 180,E1 -23671.778,E2 -23671.778} C_VEL
LIN {X 0,Y 174.577,Z 225.216,A -85,B 0,C 180,E1 -23673.266,E2 -23673.266} C_VEL
LIN {X 0,Y 169.335,Z 211.534,A -85,B 0,C 180,E1 -23675.083,E2 -23675.083} C_VEL
LIN {X 0,Y 159.342,Z 193.991,A -85,B 0,C 180,E1 -23678.392,E2 -23678.392} C_VEL
LIN {X 0,Y 157.822,Z 190.929,A -85,B 0,C 180,E1 -23679.131,E2 -23679.131} C_VEL
LIN {X 0,Y 157.744,Z 190.398,A -85,B 0,C 180,E1 -23679.62,E2 -23679.62} C_VEL
LIN {X 0,Y 157.452,Z 190.373,A -85,B 0,C 180,E1 -23685.537,E2 -23685.537} C_VEL
LIN {X 0,Y 157.37,Z 190.373,A -85,B 0,C 180,E1 -23690.935,E2 -23690.935} C_VEL
LIN {X 0,Y 157.31,Z 190.36,A -85,B 0,C 180,E1 -23696.683,E2 -23696.683} C_VEL
LIN {X 0,Y 157.275,Z 190.388,A -85,B 0,C 180,E1 -23702.43,E2 -23702.43} C_VEL
LIN {X 0,Y 157.269,Z 190.354,A -85,B 0,C 180,E1 -23706.451,E2 -23706.451} C_VEL
LIN {X 0,Y 157.212,Z 190.402,A -85,B 0,C 180,E1 -23712.113,E2 -23712.113} C_VEL
LIN {X 0,Y 157.213,Z 190.349,A -85,B 0,C 180,E1 -23717.892,E2 -23717.892} C_VEL
LIN {X 0,Y 157.269,Z 190.389,A -85,B 0,C 180,E1 -23723.554,E2 -23723.554} C_VEL
LIN {X 0,Y 157.286,Z 190.381,A -85,B 0,C 180,E1 -23728.104,E2 -23728.104} C_VEL
LIN {X 0,Y 157.313,Z 190.389,A -85,B 0,C 180,E1 -23733.466,E2 -23733.466} C_VEL
LIN {X 0,Y 157.396,Z 190.375,A -85,B 0,C 180,E1 -23739.672,E2 -23739.672} C_VEL
LIN {X 0,Y 157.445,Z 190.356,A -85,B 0,C 180,E1 -23744.466,E2 -23744.466} C_VEL
LIN {X 0,Y 157.691,Z 190.338,A -85,B 0,C 180,E1 -23749.732,E2 -23749.732} C_VEL
LIN {X 0,Y 157.762,Z 190.318,A -85,B 0,C 180,E1 -23752.321,E2 -23752.321} C_VEL
LIN {X 0,Y 158.24,Z 190.248,A -85,B 0,C 180,E1 -23760.001,E2 -23760.001} C_VEL
LIN {X 0,Y 157.764,Z 190.322,A -85,B 0,C 180,E1 -23767.681,E2 -23767.681} C_VEL
LIN {X 0,Y 157.638,Z 190.346,A -85,B 0,C 180,E1 -23771.228,E2 -23771.228} C_VEL
LIN {X 0,Y 157.42,Z 190.334,A -85,B 0,C 180,E1 -23775.539,E2 -23775.539} C_VEL
LIN {X 0,Y 157.309,Z 190.39,A -85,B 0,C 180,E1 -23780.943,E2 -23780.943} C_VEL
LIN {X 0,Y 157.272,Z 190.365,A -85,B 0,C 180,E1 -23786.649,E2 -23786.649} C_VEL
LIN {X 0,Y 157.27,Z 190.378,A -85,B 0,C 180,E1 -23792.43,E2 -23792.43} C_VEL
LIN {X 0,Y 157.264,Z 190.392,A -85,B 0,C 180,E1 -23796.444,E2 -23796.444} C_VEL
LIN {X 0,Y 157.195,Z 190.399,A -85,B 0,C 180,E1 -23802.117,E2 -23802.117} C_VEL
LIN {X 0,Y 157.251,Z 190.566,A -85,B 0,C 180,E1 -23804.244,E2 -23804.244} C_VEL
LIN {X 0,Y 157.478,Z 191.567,A -85,B 0,C 180,E1 -23804.723,E2 -23804.723} C_VEL
LIN {X 0,Y 159.193,Z 194.5,A -85,B 0,C 180,E1 -23805.384,E2 -23805.384} C_VEL
LIN {X 0,Y 163.56,Z 202.783,A -85,B 0,C 180,E1 -23806.927,E2 -23806.927} C_VEL
LIN {X 0,Y 170.977,Z 219.866,A -85,B 0,C 180,E1 -23809.506,E2 -23809.506} C_VEL
LIN {X 0,Y 177.726,Z 238.643,A -85,B 0,C 180,E1 -23811.809,E2 -23811.809} C_VEL
LIN {X 0,Y 178.742,Z 246.355,A -85,B 0,C 180,E1 -23812.389,E2 -23812.389} C_VEL
LIN {X 0,Y 175.587,Z 298.156,A -85,B 0,C 180,E1 -23814.609,E2 -23814.609} C_VEL
LIN {X 0,Y 173.872,Z 311.999,A -85,B 0,C 180,E1 -23815.621,E2 -23815.621} C_VEL
LIN {X 0,Y 171.933,Z 324.583,A -85,B 0,C 180,E1 -23817.03,E2 -23817.03} C_VEL
LIN {X 0,Y 169.574,Z 336.234,A -85,B 0,C 180,E1 -23818.795,E2 -23818.795} C_VEL
LIN {X 0,Y 167.215,Z 346.259,A -85,B 0,C 180,E1 -23820.749,E2 -23820.749} C_VEL
LIN {X 0,Y 164.526,Z 356.763,A -85,B 0,C 180,E1 -23823.348,E2 -23823.348} C_VEL
LIN {X 0,Y 162.094,Z 365.429,A -85,B 0,C 180,E1 -23826.046,E2 -23826.046} C_VEL
LIN {X 0,Y 160.08,Z 372.516,A -85,B 0,C 180,E1 -23828.762,E2 -23828.762} C_VEL
LIN {X 0,Y 158.239,Z 379.196,A -85,B 0,C 180,E1 -23831.884,E2 -23831.884} C_VEL
LIN {X 0,Y 156.405,Z 386.152,A -85,B 0,C 180,E1 -23835.987,E2 -23835.987} C_VEL
LIN {X 0,Y 155.16,Z 388.806,A -85,B 0,C 180,E1 -23837.886,E2 -23837.886} C_VEL
LIN {X 0,Y 151.582,Z 392.497,A -85,B 0,C 180,E1 -23841.064,E2 -23841.064} C_VEL
LIN {X 0,Y 148.81,Z 394.927,A -85,B 0,C 180,E1 -23843.768,E2 -23843.768} C_VEL
LIN {X 0,Y 147.649,Z 396.53,A -85,B 0,C 180,E1 -23845.935,E2 -23845.935} C_VEL
LIN {X 0,Y 147.554,Z 396.99,A -85,B 0,C 180,E1 -23846.675,E2 -23846.675} C_VEL
LIN {X 0,Y 147.6,Z 399.102,A -85,B 0,C 180,E1 -23850.636,E2 -23850.636} C_VEL
LIN {X 0,Y 147.717,Z 400.444,A -85,B 0,C 180,E1 -23855.457,E2 -23855.457} C_VEL
LIN {X 0,Y 148.02,Z 400.668,A -85,B 0,C 180,E1 -23858.186,E2 -23858.186} C_VEL
LIN {X 0,Y 148.568,Z 400.502,A -85,B 0,C 180,E1 -23860.904,E2 -23860.904} C_VEL
LIN {X 0,Y 150.589,Z 398.967,A -85,B 0,C 180,E1 -23866.258,E2 -23866.258} C_VEL
LIN {X 0,Y 151.98,Z 397.631,A -85,B 0,C 180,E1 -23868.884,E2 -23868.884} C_VEL
LIN {X 0,Y 154.863,Z 394.834,A -85,B 0,C 180,E1 -23872.687,E2 -23872.687} C_VEL
LIN {X 0,Y 158.515,Z 391.06,A -85,B 0,C 180,E1 -23876.315,E2 -23876.315} C_VEL
LIN {X 0,Y 162.433,Z 386.201,A -85,B 0,C 180,E1 -23879.875,E2 -23879.875} C_VEL
LIN {X 0,Y 167.106,Z 380.216,A -85,B 0,C 180,E1 -23883.14,E2 -23883.14} C_VEL
LIN {X 0,Y 172.438,Z 372.754,A -85,B 0,C 180,E1 -23886.222,E2 -23886.222} C_VEL
LIN {X 0,Y 177.298,Z 365.174,A -85,B 0,C 180,E1 -23888.629,E2 -23888.629} C_VEL
LIN {X 0,Y 182.36,Z 356.068,A -85,B 0,C 180,E1 -23890.928,E2 -23890.928} C_VEL
LIN {X 0,Y 187.809,Z 344.823,A -85,B 0,C 180,E1 -23893.069,E2 -23893.069} C_VEL
LIN {X 0,Y 192.424,Z 333.578,A -85,B 0,C 180,E1 -23894.67,E2 -23894.67} C_VEL
LIN {X 0,Y 196.533,Z 320.968,A -85,B 0,C 180,E1 -23895.999,E2 -23895.999} C_VEL
LIN {X 0,Y 199.93,Z 307.108,A -85,B 0,C 180,E1 -23897.034,E2 -23897.034} C_VEL
LIN {X 0,Y 202.161,Z 293.694,A -85,B 0,C 180,E1 -23897.64,E2 -23897.64} C_VEL
LIN {X 0,Y 204.803,Z 265.726,A -85,B 0,C 180,E1 -23898.666,E2 -23898.666} C_VEL
LIN {X 0,Y 202.086,Z 258.482,A -85,B 0,C 180,E1 -23900.728,E2 -23900.728} C_VEL
LIN {X 0,Y 199.067,Z 251.555,A -85,B 0,C 180,E1 -23903.233,E2 -23903.233} C_VEL
LIN {X 0,Y 196.979,Z 247.187,A -85,B 0,C 180,E1 -23905.189,E2 -23905.189} C_VEL
LIN {X 0,Y 195.009,Z 243.229,A -85,B 0,C 180,E1 -23907.275,E2 -23907.275} C_VEL
LIN {X 0,Y 193.094,Z 239.635,A -85,B 0,C 180,E1 -23909.648,E2 -23909.648} C_VEL
LIN {X 0,Y 190.604,Z 235.056,A -85,B 0,C 180,E1 -23913.738,E2 -23913.738} C_VEL
LIN {X 0,Y 189.122,Z 232.926,A -85,B 0,C 180,E1 -23917.484,E2 -23917.484} C_VEL
LIN {X 0,Y 188.466,Z 232.223,A -85,B 0,C 180,E1 -23922.642,E2 -23922.642} C_VEL
LIN {X 0,Y 189.434,Z 232.978,A -85,B 0,C 180,E1 -23927.628,E2 -23927.628} C_VEL
LIN {X 0,Y 190.487,Z 233.68,A -85,B 0,C 180,E1 -23929.99,E2 -23929.99} C_VEL
LIN {X 0,Y 192.082,Z 236.836,A -85,B 0,C 180,E1 -23932.992,E2 -23932.992} C_VEL
LIN {X 0,Y 193.791,Z 238.671,A -85,B 0,C 180,E1 -23935.219,E2 -23935.219} C_VEL
LIN {X 0,Y 196.328,Z 243.374,A -85,B 0,C 180,E1 -23938.128,E2 -23938.128} C_VEL
LIN {X 0,Y 199.173,Z 248.786,A -85,B 0,C 180,E1 -23940.842,E2 -23940.842} C_VEL
LIN {X 0,Y 202.685,Z 256.537,A -85,B 0,C 180,E1 -23943.719,E2 -23943.719} C_VEL
LIN {X 0,Y 205.12,Z 262.758,A -85,B 0,C 180,E1 -23945.535,E2 -23945.535} C_VEL
LIN {X 0,Y 201.766,Z 295.113,A -85,B 0,C 180,E1 -23946.686,E2 -23946.686} C_VEL
LIN {X 0,Y 199.241,Z 308.548,A -85,B 0,C 180,E1 -23947.442,E2 -23947.442} C_VEL
LIN {X 0,Y 196.292,Z 320.064,A -85,B 0,C 180,E1 -23948.426,E2 -23948.426} C_VEL
LIN {X 0,Y 192.11,Z 332.499,A -85,B 0,C 180,E1 -23949.866,E2 -23949.866} C_VEL
LIN {X 0,Y 187.29,Z 344.106,A -85,B 0,C 180,E1 -23951.664,E2 -23951.664} C_VEL
LIN {X 0,Y 182.271,Z 354.199,A -85,B 0,C 180,E1 -23953.741,E2 -23953.741} C_VEL
LIN {X 0,Y 177.029,Z 363.264,A -85,B 0,C 180,E1 -23956.134,E2 -23956.134} C_VEL
LIN {X 0,Y 171.175,Z 372.165,A -85,B 0,C 180,E1 -23959.22,E2 -23959.22} C_VEL
LIN {X 0,Y 166.204,Z 378.911,A -85,B 0,C 180,E1 -23962.368,E2 -23962.368} C_VEL
LIN {X 0,Y 161.649,Z 384.448,A -85,B 0,C 180,E1 -23965.769,E2 -23965.769} C_VEL
LIN {X 0,Y 157.599,Z 388.844,A -85,B 0,C 180,E1 -23969.374,E2 -23969.374} C_VEL
LIN {X 0,Y 153.327,Z 393.021,A -85,B 0,C 180,E1 -23974.412,E2 -23974.412} C_VEL
LIN {X 0,Y 151.181,Z 394.788,A -85,B 0,C 180,E1 -23977.794,E2 -23977.794} C_VEL
LIN {X 0,Y 149.497,Z 395.905,A -85,B 0,C 180,E1 -23981.226,E2 -23981.226} C_VEL
LIN {X 0,Y 148.131,Z 396.347,A -85,B 0,C 180,E1 -23985.369,E2 -23985.369} C_VEL
LIN {X 0,Y 147.297,Z 395.819,A -85,B 0,C 180,E1 -23989.764,E2 -23989.764} C_VEL
LIN {X 0,Y 147.04,Z 393.835,A -85,B 0,C 180,E1 -23995.005,E2 -23995.005} C_VEL
LIN {X 0,Y 147.414,Z 391.232,A -85,B 0,C 180,E1 -23999.107,E2 -23999.107} C_VEL
LIN {X 0,Y 148.146,Z 387.807,A -85,B 0,C 180,E1 -24002.99,E2 -24002.99} C_VEL
LIN {X 0,Y 149.252,Z 382.941,A -85,B 0,C 180,E1 -24007.144,E2 -24007.144} C_VEL
LIN {X 0,Y 151.111,Z 375.919,A -85,B 0,C 180,E1 -24011.707,E2 -24011.707} C_VEL
LIN {X 0,Y 153.33,Z 368.249,A -85,B 0,C 180,E1 -24015.565,E2 -24015.565} C_VEL
LIN {X 0,Y 156.191,Z 358.608,A -85,B 0,C 180,E1 -24019.306,E2 -24019.306} C_VEL
LIN {X 0,Y 159.074,Z 348.445,A -85,B 0,C 180,E1 -24022.386,E2 -24022.386} C_VEL
LIN {X 0,Y 161.996,Z 337.124,A -85,B 0,C 180,E1 -24025.025,E2 -24025.025} C_VEL
LIN {X 0,Y 164.751,Z 324.632,A -85,B 0,C 180,E1 -24027.252,E2 -24027.252} C_VEL
LIN {X 0,Y 166.797,Z 313.038,A -85,B 0,C 180,E1 -24028.795,E2 -24028.795} C_VEL
LIN {X 0,Y 168.691,Z 299.482,A -85,B 0,C 180,E1 -24030.055,E2 -24030.055} C_VEL
LIN {X 0,Y 169.922,Z 285.955,A -85,B 0,C 180,E1 -24030.844,E2 -24030.844} C_VEL
LIN {X 0,Y 172.764,Z 239.895,A -85,B 0,C 180,E1 -24032.815,E2 -24032.815} C_VEL
LIN {X 0,Y 169.111,Z 228.907,A -85,B 0,C 180,E1 -24034.146,E2 -24034.146} C_VEL
LIN {X 0,Y 163.911,Z 215.167,A -85,B 0,C 180,E1 -24036.041,E2 -24036.041} C_VEL
LIN {X 0,Y 154.097,Z 197.921,A -85,B 0,C 180,E1 -24039.499,E2 -24039.499} C_VEL
LIN {X 0,Y 152.323,Z 194.978,A -85,B 0,C 180,E1 -24040.16,E2 -24040.16} C_VEL
LIN {X 0,Y 150.807,Z 192.178,A -85,B 0,C 180,E1 -24040.827,E2 -24040.827} C_VEL
LIN {X 0,Y 150.581,Z 191.314,A -85,B 0,C 180,E1 -24041.449,E2 -24041.449} C_VEL
LIN {X 0,Y 150.36,Z 191.252,A -85,B 0,C 180,E1 -24046.29,E2 -24046.29} C_VEL
LIN {X 0,Y 150.351,Z 191.244,A -85,B 0,C 180,E1 -24050.795,E2 -24050.795} C_VEL
LIN {X 0,Y 150.242,Z 191.241,A -85,B 0,C 180,E1 -24057.282,E2 -24057.282} C_VEL
LIN {X 0,Y 150.215,Z 191.265,A -85,B 0,C 180,E1 -24062.634,E2 -24062.634} C_VEL
LIN {X 0,Y 150.174,Z 191.241,A -85,B 0,C 180,E1 -24067.476,E2 -24067.476} C_VEL
LIN {X 0,Y 150.152,Z 191.282,A -85,B 0,C 180,E1 -24071.507,E2 -24071.507} C_VEL
LIN {X 0,Y 150.127,Z 191.255,A -85,B 0,C 180,E1 -24075.398,E2 -24075.398} C_VEL
LIN {X 0,Y 150.151,Z 191.227,A -85,B 0,C 180,E1 -24079.06,E2 -24079.06} C_VEL
LIN {X 0,Y 150.181,Z 191.264,A -85,B 0,C 180,E1 -24082.71,E2 -24082.71} C_VEL
LIN {X 0,Y 150.211,Z 191.267,A -85,B 0,C 180,E1 -24087.374,E2 -24087.374} C_VEL
LIN {X 0,Y 150.242,Z 191.271,A -85,B 0,C 180,E1 -24092.725,E2 -24092.725} C_VEL
LIN {X 0,Y 150.353,Z 191.252,A -85,B 0,C 180,E1 -24099.212,E2 -24099.212} C_VEL
LIN {X 0,Y 150.356,Z 191.24,A -85,B 0,C 180,E1 -24103.714,E2 -24103.714} C_VEL
LIN {X 0,Y 150.614,Z 191.222,A -85,B 0,C 180,E1 -24109.244,E2 -24109.244} C_VEL
LIN {X 0,Y 150.685,Z 191.199,A -85,B 0,C 180,E1 -24111.958,E2 -24111.958} C_VEL
LIN {X 0,Y 151.201,Z 191.122,A -85,B 0,C 180,E1 -24120.001,E2 -24120.001} C_VEL
LIN {X 0,Y 150.703,Z 191.204,A -85,B 0,C 180,E1 -24128.044,E2 -24128.044} C_VEL
LIN {X 0,Y 150.58,Z 191.223,A -85,B 0,C 180,E1 -24131.431,E2 -24131.431} C_VEL
LIN {X 0,Y 150.323,Z 191.216,A -85,B 0,C 180,E1 -24136.292,E2 -24136.292} C_VEL
LIN {X 0,Y 150.287,Z 191.264,A -85,B 0,C 180,E1 -24140.722,E2 -24140.722} C_VEL
LIN {X 0,Y 150.19,Z 191.249,A -85,B 0,C 180,E1 -24147.237,E2 -24147.237} C_VEL
LIN {X 0,Y 150.211,Z 191.254,A -85,B 0,C 180,E1 -24152.625,E2 -24152.625} C_VEL
LIN {X 0,Y 150.175,Z 191.279,A -85,B 0,C 180,E1 -24157.474,E2 -24157.474} C_VEL
LIN {X 0,Y 150.192,Z 191.487,A -85,B 0,C 180,E1 -24162.382,E2 -24162.382} C_VEL
LIN {X 0,Y 150.471,Z 192.525,A -85,B 0,C 180,E1 -24162.903,E2 -24162.903} C_VEL
LIN {X 0,Y 152.095,Z 195.314,A -85,B 0,C 180,E1 -24163.568,E2 -24163.568} C_VEL
LIN {X 0,Y 157.747,Z 205.306,A -85,B 0,C 180,E1 -24165.696,E2 -24165.696} C_VEL
LIN {X 0,Y 165.362,Z 223.117,A -85,B 0,C 180,E1 -24168.512,E2 -24168.512} C_VEL
LIN {X 0,Y 171.872,Z 241.442,A -85,B 0,C 180,E1 -24170.876,E2 -24170.876} C_VEL
LIN {X 0,Y 172.482,Z 247.404,A -85,B 0,C 180,E1 -24171.315,E2 -24171.315} C_VEL
LIN {X 0,Y 169.238,Z 298.129,A -85,B 0,C 180,E1 -24173.554,E2 -24173.554} C_VEL
LIN {X 0,Y 167.496,Z 311.758,A -85,B 0,C 180,E1 -24174.578,E2 -24174.578} C_VEL
LIN {X 0,Y 165.581,Z 323.886,A -85,B 0,C 180,E1 -24175.96,E2 -24175.96} C_VEL
LIN {X 0,Y 163.129,Z 335.658,A -85,B 0,C 180,E1 -24177.779,E2 -24177.779} C_VEL
LIN {X 0,Y 160.674,Z 345.768,A -85,B 0,C 180,E1 -24179.798,E2 -24179.798} C_VEL
LIN {X 0,Y 157.87,Z 356.338,A -85,B 0,C 180,E1 -24182.49,E2 -24182.49} C_VEL
LIN {X 0,Y 155.271,Z 365.163,A -85,B 0,C 180,E1 -24185.322,E2 -24185.322} C_VEL
LIN {X 0,Y 152.997,Z 372.935,A -85,B 0,C 180,E1 -24188.437,E2 -24188.437} C_VEL
LIN {X 0,Y 150.725,Z 380.675,A -85,B 0,C 180,E1 -24192.355,E2 -24192.355} C_VEL
LIN {X 0,Y 149.14,Z 386.882,A -85,B 0,C 180,E1 -24196.369,E2 -24196.369} C_VEL
LIN {X 0,Y 148.15,Z 391.775,A -85,B 0,C 180,E1 -24200.44,E2 -24200.44} C_VEL
LIN {X 0,Y 147.671,Z 395.497,A -85,B 0,C 180,E1 -24204.535,E2 -24204.535} C_VEL
LIN {X 0,Y 147.554,Z 396.99,A -85,B 0,C 180,E1 -24206.675,E2 -24206.675} C_VEL
LIN {X 0,Y 146.868,Z 398.353,A -85,B 0,C 180,E1 -24208.892,E2 -24208.892} C_VEL
LIN {X 0,Y 145.287,Z 399.358,A -85,B 0,C 180,E1 -24211.106,E2 -24211.106} C_VEL
LIN {X 0,Y 141.771,Z 400.41,A -85,B 0,C 180,E1 -24215.682,E2 -24215.682} C_VEL
LIN {X 0,Y 141.002,Z 400.531,A -85,B 0,C 180,E1 -24218.094,E2 -24218.094} C_VEL
LIN {X 0,Y 141.044,Z 400.517,A -85,B 0,C 180,E1 -24218.906,E2 -24218.906} C_VEL
LIN {X 0,Y 142.533,Z 399.951,A -85,B 0,C 180,E1 -24224.27,E2 -24224.27} C_VEL
LIN {X 0,Y 145.26,Z 397.785,A -85,B 0,C 180,E1 -24229.793,E2 -24229.793} C_VEL
LIN {X 0,Y 148.331,Z 395.128,A -85,B 0,C 180,E1 -24233.746,E2 -24233.746} C_VEL
LIN {X 0,Y 152.201,Z 391.493,A -85,B 0,C 180,E1 -24237.497,E2 -24237.497} C_VEL
LIN {X 0,Y 157.466,Z 385.483,A -85,B 0,C 180,E1 -24242.003,E2 -24242.003} C_VEL
LIN {X 0,Y 163.063,Z 378.711,A -85,B 0,C 180,E1 -24245.577,E2 -24245.577} C_VEL
LIN {X 0,Y 168.718,Z 370.934,A -85,B 0,C 180,E1 -24248.666,E2 -24248.666} C_VEL
LIN {X 0,Y 173.923,Z 363.051,A -85,B 0,C 180,E1 -24251.04,E2 -24251.04} C_VEL
LIN {X 0,Y 179.399,Z 353.52,A -85,B 0,C 180,E1 -24253.276,E2 -24253.276} C_VEL
LIN {X 0,Y 184.589,Z 343.014,A -85,B 0,C 180,E1 -24255.16,E2 -24255.16} C_VEL
LIN {X 0,Y 189.35,Z 331.254,A -85,B 0,C 180,E1 -24256.749,E2 -24256.749} C_VEL
LIN {X 0,Y 193.392,Z 318.902,A -85,B 0,C 180,E1 -24257.959,E2 -24257.959} C_VEL
LIN {X 0,Y 196.573,Z 305.796,A -85,B 0,C 180,E1 -24258.877,E2 -24258.877} C_VEL
LIN {X 0,Y 198.825,Z 292.201,A -85,B 0,C 180,E1 -24259.455,E2 -24259.455} C_VEL
LIN {X 0,Y 201.156,Z 268.814,A -85,B 0,C 180,E1 -24260.305,E2 -24260.305} C_VEL
LIN {X 0,Y 198.283,Z 261.021,A -85,B 0,C 180,E1 -24262.767,E2 -24262.767} C_VEL
LIN {X 0,Y 195.378,Z 254.235,A -85,B 0,C 180,E1 -24265.577,E2 -24265.577} C_VEL
LIN {X 0,Y 192.909,Z 249.065,A -85,B 0,C 180,E1 -24268.359,E2 -24268.359} C_VEL
LIN {X 0,Y 191.486,Z 246.14,A -85,B 0,C 180,E1 -24270.345,E2 -24270.345} C_VEL
LIN {X 0,Y 189.35,Z 241.925,A -85,B 0,C 180,E1 -24274.143,E2 -24274.143} C_VEL
LIN {X 0,Y 187.948,Z 239.822,A -85,B 0,C 180,E1 -24278.041,E2 -24278.041} C_VEL
LIN {X 0,Y 187.431,Z 239.255,A -85,B 0,C 180,E1 -24282.543,E2 -24282.543} C_VEL
LIN {X 0,Y 188.374,Z 239.974,A -85,B 0,C 180,E1 -24287.557,E2 -24287.557} C_VEL
LIN {X 0,Y 189.229,Z 240.584,A -85,B 0,C 180,E1 -24289.559,E2 -24289.559} C_VEL
LIN {X 0,Y 190.831,Z 243.796,A -85,B 0,C 180,E1 -24292.738,E2 -24292.738} C_VEL
LIN {X 0,Y 192.3,Z 245.495,A -85,B 0,C 180,E1 -24294.737,E2 -24294.737} C_VEL
LIN {X 0,Y 194.394,Z 249.69,A -85,B 0,C 180,E1 -24297.339,E2 -24297.339} C_VEL
LIN {X 0,Y 196.937,Z 254.766,A -85,B 0,C 180,E1 -24299.949,E2 -24299.949} C_VEL
LIN {X 0,Y 200.12,Z 262.317,A -85,B 0,C 180,E1 -24302.777,E2 -24302.777} C_VEL
LIN {X 0,Y 201.442,Z 265.847,A -85,B 0,C 180,E1 -24303.871,E2 -24303.871} C_VEL
LIN {X 0,Y 198.291,Z 294.903,A -85,B 0,C 180,E1 -24304.911,E2 -24304.911} C_VEL
LIN {X 0,Y 195.556,Z 308.877,A -85,B 0,C 180,E1 -24305.683,E2 -24305.683} C_VEL
LIN {X 0,Y 192.131,Z 321.459,A -85,B 0,C 180,E1 -24306.773,E2 -24306.773} C_VEL
LIN {X 0,Y 187.821,Z 333.601,A -85,B 0,C 180,E1 -24308.201,E2 -24308.201} C_VEL
LIN {X 0,Y 182.84,Z 344.907,A -85,B 0,C 180,E1 -24309.969,E2 -24309.969} C_VEL
LIN {X 0,Y 177.096,Z 355.781,A -85,B 0,C 180,E1 -24312.264,E2 -24312.264} C_VEL
LIN {X 0,Y 171.906,Z 364.183,A -85,B 0,C 180,E1 -24314.56,E2 -24314.56} C_VEL
LIN {X 0,Y 165.897,Z 372.698,A -85,B 0,C 180,E1 -24317.602,E2 -24317.602} C_VEL
LIN {X 0,Y 160.109,Z 379.954,A -85,B 0,C 180,E1 -24321.139,E2 -24321.139} C_VEL
LIN {X 0,Y 154.993,Z 385.693,A -85,B 0,C 180,E1 -24324.931,E2 -24324.931} C_VEL
LIN {X 0,Y 151.361,Z 389.281,A -85,B 0,C 180,E1 -24328.098,E2 -24328.098} C_VEL
LIN {X 0,Y 146.898,Z 393.258,A -85,B 0,C 180,E1 -24333.156,E2 -24333.156} C_VEL
LIN {X 0,Y 143.58,Z 395.589,A -85,B 0,C 180,E1 -24338.454,E2 -24338.454} C_VEL
LIN {X 0,Y 141.327,Z 396.452,A -85,B 0,C 180,E1 -24344.121,E2 -24344.121} C_VEL
LIN {X 0,Y 140.261,Z 395.864,A -85,B 0,C 180,E1 -24349.359,E2 -24349.359} C_VEL
LIN {X 0,Y 139.915,Z 394.456,A -85,B 0,C 180,E1 -24353.482,E2 -24353.482} C_VEL
LIN {X 0,Y 140.227,Z 391.666,A -85,B 0,C 180,E1 -24358.429,E2 -24358.429} C_VEL
LIN {X 0,Y 141.176,Z 387.211,A -85,B 0,C 180,E1 -24363.644,E2 -24363.644} C_VEL
LIN {X 0,Y 142.413,Z 382.064,A -85,B 0,C 180,E1 -24368.071,E2 -24368.071} C_VEL
LIN {X 0,Y 144.166,Z 375.771,A -85,B 0,C 180,E1 -24372.264,E2 -24372.264} C_VEL
LIN {X 0,Y 146.404,Z 368.425,A -85,B 0,C 180,E1 -24376.115,E2 -24376.115} C_VEL
LIN {X 0,Y 149.228,Z 359.291,A -85,B 0,C 180,E1 -24379.846,E2 -24379.846} C_VEL
LIN {X 0,Y 152.159,Z 349.321,A -85,B 0,C 180,E1 -24383.039,E2 -24383.039} C_VEL
LIN {X 0,Y 155.061,Z 338.883,A -85,B 0,C 180,E1 -24385.643,E2 -24385.643} C_VEL
LIN {X 0,Y 157.637,Z 327.924,A -85,B 0,C 180,E1 -24387.767,E2 -24387.767} C_VEL
LIN {X 0,Y 159.936,Z 316.028,A -85,B 0,C 180,E1 -24389.531,E2 -24389.531} C_VEL
LIN {X 0,Y 161.948,Z 302.866,A -85,B 0,C 180,E1 -24390.935,E2 -24390.935} C_VEL
LIN {X 0,Y 163.469,Z 288.93,A -85,B 0,C 180,E1 -24391.854,E2 -24391.854} C_VEL
LIN {X 0,Y 166.487,Z 240.838,A -85,B 0,C 180,E1 -24394.009,E2 -24394.009} C_VEL
LIN {X 0,Y 161.409,Z 226.507,A -85,B 0,C 180,E1 -24395.93,E2 -24395.93} C_VEL
LIN {X 0,Y 158.425,Z 218.606,A -85,B 0,C 180,E1 -24397.095,E2 -24397.095} C_VEL
LIN {X 0,Y 147.955,Z 200.095,A -85,B 0,C 180,E1 -24401.024,E2 -24401.024} C_VEL
LIN {X 0,Y 145.218,Z 195.988,A -85,B 0,C 180,E1 -24402.112,E2 -24402.112} C_VEL
LIN {X 0,Y 143.638,Z 193.195,A -85,B 0,C 180,E1 -24402.866,E2 -24402.866} C_VEL
LIN {X 0,Y 143.398,Z 192.22,A -85,B 0,C 180,E1 -24403.537,E2 -24403.537} C_VEL
LIN {X 0,Y 143.299,Z 192.115,A -85,B 0,C 180,E1 -24410.081,E2 -24410.081} C_VEL
LIN {X 0,Y 143.156,Z 192.121,A -85,B 0,C 180,E1 -24416.224,E2 -24416.224} C_VEL
LIN {X 0,Y 143.121,Z 192.148,A -85,B 0,C 180,E1 -24419.413,E2 -24419.413} C_VEL
LIN {X 0,Y 143.144,Z 192.132,A -85,B 0,C 180,E1 -24423.422,E2 -24423.422} C_VEL
LIN {X 0,Y 143.062,Z 192.151,A -85,B 0,C 180,E1 -24429.693,E2 -24429.693} C_VEL
LIN {X 0,Y 143.058,Z 192.159,A -85,B 0,C 180,E1 -24433.458,E2 -24433.458} C_VEL
LIN {X 0,Y 143.048,Z 192.111,A -85,B 0,C 180,E1 -24437.476,E2 -24437.476} C_VEL
LIN {X 0,Y 143.079,Z 192.135,A -85,B 0,C 180,E1 -24441.809,E2 -24441.809} C_VEL
LIN {X 0,Y 143.179,Z 192.142,A -85,B 0,C 180,E1 -24447.322,E2 -24447.322} C_VEL
LIN {X 0,Y 143.186,Z 192.148,A -85,B 0,C 180,E1 -24452.071,E2 -24452.071} C_VEL
LIN {X 0,Y 143.279,Z 192.128,A -85,B 0,C 180,E1 -24458.75,E2 -24458.75} C_VEL
LIN {X 0,Y 143.299,Z 192.125,A -85,B 0,C 180,E1 -24462.888,E2 -24462.888} C_VEL
LIN {X 0,Y 143.541,Z 192.103,A -85,B 0,C 180,E1 -24468.707,E2 -24468.707} C_VEL
LIN {X 0,Y 143.611,Z 192.081,A -85,B 0,C 180,E1 -24471.559,E2 -24471.559} C_VEL
LIN {X 0,Y 144.159,Z 191.997,A -85,B 0,C 180,E1 -24480.001,E2 -24480.001} C_VEL
LIN {X 0,Y 143.625,Z 192.088,A -85,B 0,C 180,E1 -24488.443,E2 -24488.443} C_VEL
LIN {X 0,Y 143.506,Z 192.103,A -85,B 0,C 180,E1 -24491.619,E2 -24491.619} C_VEL
LIN {X 0,Y 143.262,Z 192.098,A -85,B 0,C 180,E1 -24497.119,E2 -24497.119} C_VEL
LIN {X 0,Y 143.224,Z 192.145,A -85,B 0,C 180,E1 -24501.194,E2 -24501.194} C_VEL
LIN {X 0,Y 143.147,Z 192.131,A -85,B 0,C 180,E1 -24507.899,E2 -24507.899} C_VEL
LIN {X 0,Y 143.141,Z 192.13,A -85,B 0,C 180,E1 -24513.414,E2 -24513.414} C_VEL
LIN {X 0,Y 143.086,Z 192.195,A -85,B 0,C 180,E1 -24520.013,E2 -24520.013} C_VEL
LIN {X 0,Y 143.217,Z 192.902,A -85,B 0,C 180,E1 -24520.714,E2 -24520.714} C_VEL
LIN {X 0,Y 144.753,Z 195.899,A -85,B 0,C 180,E1 -24521.514,E2 -24521.514} C_VEL
LIN {X 0,Y 145.943,Z 197.728,A -85,B 0,C 180,E1 -24521.999,E2 -24521.999} C_VEL
LIN {X 0,Y 152.553,Z 209.144,A -85,B 0,C 180,E1 -24524.609,E2 -24524.609} C_VEL
LIN {X 0,Y 159.801,Z 226.414,A -85,B 0,C 180,E1 -24527.478,E2 -24527.478} C_VEL
LIN {X 0,Y 165.895,Z 243.675,A -85,B 0,C 180,E1 -24529.809,E2 -24529.809} C_VEL
LIN {X 0,Y 166.287,Z 248.754,A -85,B 0,C 180,E1 -24530.178,E2 -24530.178} C_VEL
LIN {X 0,Y 162.995,Z 297.733,A -85,B 0,C 180,E1 -24532.394,E2 -24532.394} C_VEL
LIN {X 0,Y 161.19,Z 311.524,A -85,B 0,C 180,E1 -24533.455,E2 -24533.455} C_VEL
LIN {X 0,Y 159.083,Z 324.185,A -85,B 0,C 180,E1 -24534.946,E2 -24534.946} C_VEL
LIN {X 0,Y 156.321,Z 336.649,A -85,B 0,C 180,E1 -24536.964,E2 -24536.964} C_VEL
LIN {X 0,Y 153.526,Z 347.887,A -85,B 0,C 180,E1 -24539.382,E2 -24539.382} C_VEL
LIN {X 0,Y 150.625,Z 357.99,A -85,B 0,C 180,E1 -24542.184,E2 -24542.184} C_VEL
LIN {X 0,Y 148.345,Z 365.488,A -85,B 0,C 180,E1 -24544.759,E2 -24544.759} C_VEL
LIN {X 0,Y 145.945,Z 373.319,A -85,B 0,C 180,E1 -24548.084,E2 -24548.084} C_VEL
LIN {X 0,Y 143.616,Z 380.957,A -85,B 0,C 180,E1 -24552.188,E2 -24552.188} C_VEL
LIN {X 0,Y 141.783,Z 387.995,A -85,B 0,C 180,E1 -24557.108,E2 -24557.108} C_VEL
LIN {X 0,Y 140.906,Z 392.608,A -85,B 0,C 180,E1 -24561.392,E2 -24561.392} C_VEL
LIN {X 0,Y 140.611,Z 395.019,A -85,B 0,C 180,E1 -24564.26,E2 -24564.26} C_VEL
LIN {X 0,Y 140.484,Z 396.979,A -85,B 0,C 180,E1 -24567.13,E2 -24567.13} C_VEL
LIN {X 0,Y 140.563,Z 398.515,A -85,B 0,C 180,E1 -24569.997,E2 -24569.997} C_VEL
LIN {X 0,Y 140.492,Z 399.583,A -85,B 0,C 180,E1 -24572.864,E2 -24572.864} C_VEL
LIN {X 0,Y 140.644,Z 400.246,A -85,B 0,C 180,E1 -24575.733,E2 -24575.733} C_VEL
LIN {X 0,Y 141.044,Z 400.517,A -85,B 0,C 180,E1 -24578.906,E2 -24578.906} C_VEL
LIN {X 0,Y 140.87,Z 400.447,A -85,B 0,C 180,E1 -24581.309,E2 -24581.309} C_VEL
LIN {X 0,Y 139.275,Z 399.785,A -85,B 0,C 180,E1 -24585.312,E2 -24585.312} C_VEL
LIN {X 0,Y 138.367,Z 398.573,A -85,B 0,C 180,E1 -24589.358,E2 -24589.358} C_VEL
LIN {X 0,Y 139.248,Z 397.421,A -85,B 0,C 180,E1 -24591.721,E2 -24591.721} C_VEL
LIN {X 0,Y 143.16,Z 394.357,A -85,B 0,C 180,E1 -24596.217,E2 -24596.217} C_VEL
LIN {X 0,Y 147.404,Z 390.509,A -85,B 0,C 180,E1 -24600.037,E2 -24600.037} C_VEL
LIN {X 0,Y 151.956,Z 385.645,A -85,B 0,C 180,E1 -24603.707,E2 -24603.707} C_VEL
LIN {X 0,Y 157.397,Z 379.548,A -85,B 0,C 180,E1 -24607.066,E2 -24607.066} C_VEL
LIN {X 0,Y 163.32,Z 372.033,A -85,B 0,C 180,E1 -24610.198,E2 -24610.198} C_VEL
LIN {X 0,Y 168.721,Z 364.386,A -85,B 0,C 180,E1 -24612.597,E2 -24612.597} C_VEL
LIN {X 0,Y 174.979,Z 354.096,A -85,B 0,C 180,E1 -24615.06,E2 -24615.06} C_VEL
LIN {X 0,Y 179.712,Z 345.032,A -85,B 0,C 180,E1 -24616.745,E2 -24616.745} C_VEL
LIN {X 0,Y 184.704,Z 333.928,A -85,B 0,C 180,E1 -24618.304,E2 -24618.304} C_VEL
LIN {X 0,Y 188.834,Z 322.538,A -85,B 0,C 180,E1 -24619.516,E2 -24619.516} C_VEL
LIN {X 0,Y 192.495,Z 309.271,A -85,B 0,C 180,E1 -24620.519,E2 -24620.519} C_VEL
LIN {X 0,Y 194.946,Z 296.881,A -85,B 0,C 180,E1 -24621.133,E2 -24621.133} C_VEL
LIN {X 0,Y 197.741,Z 272.07,A -85,B 0,C 180,E1 -24621.997,E2 -24621.997} C_VEL
LIN {X 0,Y 195.131,Z 264.873,A -85,B 0,C 180,E1 -24624.498,E2 -24624.498} C_VEL
LIN {X 0,Y 192.939,Z 259.476,A -85,B 0,C 180,E1 -24626.903,E2 -24626.903} C_VEL
LIN {X 0,Y 191.107,Z 255.297,A -85,B 0,C 180,E1 -24629.235,E2 -24629.235} C_VEL
LIN {X 0,Y 189.792,Z 252.486,A -85,B 0,C 180,E1 -24631.223,E2 -24631.223} C_VEL
LIN {X 0,Y 188.054,Z 248.702,A -85,B 0,C 180,E1 -24634.678,E2 -24634.678} C_VEL
LIN {X 0,Y 186.945,Z 246.884,A -85,B 0,C 180,E1 -24637.917,E2 -24637.917} C_VEL
LIN {X 0,Y 186.4,Z 246.268,A -85,B 0,C 180,E1 -24642.443,E2 -24642.443} C_VEL
LIN {X 0,Y 187.262,Z 246.948,A -85,B 0,C 180,E1 -24647.351,E2 -24647.351} C_VEL
LIN {X 0,Y 188.022,Z 247.571,A -85,B 0,C 180,E1 -24649.228,E2 -24649.228} C_VEL
LIN {X 0,Y 189.742,Z 250.929,A -85,B 0,C 180,E1 -24652.716,E2 -24652.716} C_VEL
LIN {X 0,Y 190.746,Z 252.125,A -85,B 0,C 180,E1 -24654.13,E2 -24654.13} C_VEL
LIN {X 0,Y 192.472,Z 255.919,A -85,B 0,C 180,E1 -24656.501,E2 -24656.501} C_VEL
LIN {X 0,Y 194.839,Z 260.928,A -85,B 0,C 180,E1 -24659.103,E2 -24659.103} C_VEL
LIN {X 0,Y 197.795,Z 268.592,A -85,B 0,C 180,E1 -24661.978,E2 -24661.978} C_VEL
LIN {X 0,Y 198.014,Z 269.249,A -85,B 0,C 180,E1 -24662.179,E2 -24662.179} C_VEL
LIN {X 0,Y 194.941,Z 295.677,A -85,B 0,C 180,E1 -24663.098,E2 -24663.098} C_VEL
LIN {X 0,Y 192.21,Z 309.092,A -85,B 0,C 180,E1 -24663.837,E2 -24663.837} C_VEL
LIN {X 0,Y 188.675,Z 321.49,A -85,B 0,C 180,E1 -24664.89,E2 -24664.89} C_VEL
LIN {X 0,Y 184.66,Z 332.474,A -85,B 0,C 180,E1 -24666.152,E2 -24666.152} C_VEL
LIN {X 0,Y 179.952,Z 342.955,A -85,B 0,C 180,E1 -24667.711,E2 -24667.711} C_VEL
LIN {X 0,Y 174.516,Z 353.221,A -85,B 0,C 180,E1 -24669.719,E2 -24669.719} C_VEL
LIN {X 0,Y 168.894,Z 362.23,A -85,B 0,C 180,E1 -24672.008,E2 -24672.008} C_VEL
LIN {X 0,Y 162.383,Z 371.237,A -85,B 0,C 180,E1 -24675.05,E2 -24675.05} C_VEL
LIN {X 0,Y 156.447,Z 378.439,A -85,B 0,C 180,E1 -24678.327,E2 -24678.327} C_VEL
LIN {X 0,Y 151.229,Z 384.107,A -85,B 0,C 180,E1 -24681.824,E2 -24681.824} C_VEL
LIN {X 0,Y 146.487,Z 388.629,A -85,B 0,C 180,E1 -24685.58,E2 -24685.58} C_VEL
LIN {X 0,Y 142.431,Z 392.073,A -85,B 0,C 180,E1 -24689.565,E2 -24689.565} C_VEL
LIN {X 0,Y 139.107,Z 394.501,A -85,B 0,C 180,E1 -24693.761,E2 -24693.761} C_VEL
LIN {X 0,Y 136.005,Z 396.203,A -85,B 0,C 180,E1 -24699.19,E2 -24699.19} C_VEL
LIN {X 0,Y 134.512,Z 396.569,A -85,B 0,C 180,E1 -24702.996,E2 -24702.996} C_VEL
LIN {X 0,Y 133.392,Z 396.171,A -85,B 0,C 180,E1 -24707.527,E2 -24707.527} C_VEL
LIN {X 0,Y 132.84,Z 394.722,A -85,B 0,C 180,E1 -24712.52,E2 -24712.52} C_VEL
LIN {X 0,Y 133.074,Z 391.782,A -85,B 0,C 180,E1 -24718.125,E2 -24718.125} C_VEL
LIN {X 0,Y 133.926,Z 387.796,A -85,B 0,C 180,E1 -24723.136,E2 -24723.136} C_VEL
LIN {X 0,Y 135.209,Z 382.695,A -85,B 0,C 180,E1 -24727.865,E2 -24727.865} C_VEL
LIN {X 0,Y 137.2,Z 375.67,A -85,B 0,C 180,E1 -24732.821,E2 -24732.821} C_VEL
LIN {X 0,Y 139.588,Z 368.147,A -85,B 0,C 180,E1 -24736.908,E2 -24736.908} C_VEL
LIN {X 0,Y 142.645,Z 358.702,A -85,B 0,C 180,E1 -24740.879,E2 -24740.879} C_VEL
LIN {X 0,Y 145.646,Z 348.849,A -85,B 0,C 180,E1 -24744.118,E2 -24744.118} C_VEL
LIN {X 0,Y 148.744,Z 337.901,A -85,B 0,C 180,E1 -24746.888,E2 -24746.888} C_VEL
LIN {X 0,Y 151.817,Z 325.147,A -85,B 0,C 180,E1 -24749.34,E2 -24749.34} C_VEL
LIN {X 0,Y 154.066,Z 313.32,A -85,B 0,C 180,E1 -24751.032,E2 -24751.032} C_VEL
LIN {X 0,Y 156.127,Z 299.646,A -85,B 0,C 180,E1 -24752.381,E2 -24752.381} C_VEL
LIN {X 0,Y 157.474,Z 285.886,A -85,B 0,C 180,E1 -24753.225,E2 -24753.225} C_VEL
LIN {X 0,Y 160.275,Z 242.269,A -85,B 0,C 180,E1 -24755.234,E2 -24755.234} C_VEL
LIN {X 0,Y 153.157,Z 222.415,A -85,B 0,C 180,E1 -24758.148,E2 -24758.148} C_VEL
LIN {X 0,Y 143.272,Z 204.764,A -85,B 0,C 180,E1 -24762.079,E2 -24762.079} C_VEL
LIN {X 0,Y 139.026,Z 198.034,A -85,B 0,C 180,E1 -24763.936,E2 -24763.936} C_VEL
LIN {X 0,Y 136.738,Z 194.82,A -85,B 0,C 180,E1 -24764.984,E2 -24764.984} C_VEL
LIN {X 0,Y 136.299,Z 193.408,A -85,B 0,C 180,E1 -24765.518,E2 -24765.518} C_VEL
LIN {X 0,Y 136.233,Z 193.017,A -85,B 0,C 180,E1 -24766.486,E2 -24766.486} C_VEL
LIN {X 0,Y 136.198,Z 193.016,A -85,B 0,C 180,E1 -24771.751,E2 -24771.751} C_VEL
LIN {X 0,Y 136.099,Z 193.01,A -85,B 0,C 180,E1 -24778.618,E2 -24778.618} C_VEL
LIN {X 0,Y 136.043,Z 193,A -85,B 0,C 180,E1 -24784.632,E2 -24784.632} C_VEL
LIN {X 0,Y 136.033,Z 193.017,A -85,B 0,C 180,E1 -24789.201,E2 -24789.201} C_VEL
LIN {X 0,Y 135.999,Z 193.035,A -85,B 0,C 180,E1 -24793.66,E2 -24793.66} C_VEL
LIN {X 0,Y 135.992,Z 192.987,A -85,B 0,C 180,E1 -24797.793,E2 -24797.793} C_VEL
LIN {X 0,Y 136.028,Z 193.008,A -85,B 0,C 180,E1 -24801.686,E2 -24801.686} C_VEL
LIN {X 0,Y 136.056,Z 193.037,A -85,B 0,C 180,E1 -24805.743,E2 -24805.743} C_VEL
LIN {X 0,Y 136.143,Z 193.026,A -85,B 0,C 180,E1 -24812.317,E2 -24812.317} C_VEL
LIN {X 0,Y 136.245,Z 193.004,A -85,B 0,C 180,E1 -24818.835,E2 -24818.835} C_VEL
LIN {X 0,Y 136.268,Z 192.992,A -85,B 0,C 180,E1 -24825.057,E2 -24825.057} C_VEL
LIN {X 0,Y 136.435,Z 192.989,A -85,B 0,C 180,E1 -24828.17,E2 -24828.17} C_VEL
LIN {X 0,Y 136.541,Z 192.963,A -85,B 0,C 180,E1 -24831.118,E2 -24831.118} C_VEL
LIN {X 0,Y 137.116,Z 192.871,A -85,B 0,C 180,E1 -24840.001,E2 -24840.001} C_VEL
LIN {X 0,Y 136.552,Z 192.973,A -85,B 0,C 180,E1 -24848.884,E2 -24848.884} C_VEL
LIN {X 0,Y 136.42,Z 192.981,A -85,B 0,C 180,E1 -24851.893,E2 -24851.893} C_VEL
LIN {X 0,Y 136.172,Z 192.988,A -85,B 0,C 180,E1 -24858.04,E2 -24858.04} C_VEL
LIN {X 0,Y 136.149,Z 193.025,A -85,B 0,C 180,E1 -24861.689,E2 -24861.689} C_VEL
LIN {X 0,Y 136.067,Z 193.019,A -85,B 0,C 180,E1 -24868.585,E2 -24868.585} C_VEL
LIN {X 0,Y 136.045,Z 193.014,A -85,B 0,C 180,E1 -24874.63,E2 -24874.63} C_VEL
LIN {X 0,Y 136.068,Z 193.303,A -85,B 0,C 180,E1 -24878.127,E2 -24878.127} C_VEL
LIN {X 0,Y 136.245,Z 194.059,A -85,B 0,C 180,E1 -24878.552,E2 -24878.552} C_VEL
LIN {X 0,Y 137.638,Z 196.751,A -85,B 0,C 180,E1 -24879.28,E2 -24879.28} C_VEL
LIN {X 0,Y 138.89,Z 198.5,A -85,B 0,C 180,E1 -24879.839,E2 -24879.839} C_VEL
LIN {X 0,Y 144.81,Z 208.234,A -85,B 0,C 180,E1 -24882.404,E2 -24882.404} C_VEL
LIN {X 0,Y 148.601,Z 215.752,A -85,B 0,C 180,E1 -24883.985,E2 -24883.985} C_VEL
LIN {X 0,Y 155.213,Z 232.156,A -85,B 0,C 180,E1 -24886.761,E2 -24886.761} C_VEL
LIN {X 0,Y 159.998,Z 246.214,A -85,B 0,C 180,E1 -24888.714,E2 -24888.714} C_VEL
LIN {X 0,Y 160.017,Z 251.603,A -85,B 0,C 180,E1 -24889.04,E2 -24889.04} C_VEL
LIN {X 0,Y 156.722,Z 298.02,A -85,B 0,C 180,E1 -24891.211,E2 -24891.211} C_VEL
LIN {X 0,Y 154.852,Z 311.774,A -85,B 0,C 180,E1 -24892.315,E2 -24892.315} C_VEL
LIN {X 0,Y 152.86,Z 323.281,A -85,B 0,C 180,E1 -24893.702,E2 -24893.702} C_VEL
LIN {X 0,Y 150.414,Z 334.349,A -85,B 0,C 180,E1 -24895.488,E2 -24895.488} C_VEL
LIN {X 0,Y 147.743,Z 344.643,A -85,B 0,C 180,E1 -24897.643,E2 -24897.643} C_VEL
LIN {X 0,Y 144.679,Z 355.359,A -85,B 0,C 180,E1 -24900.536,E2 -24900.536} C_VEL
LIN {X 0,Y 141.835,Z 364.096,A -85,B 0,C 180,E1 -24903.513,E2 -24903.513} C_VEL
LIN {X 0,Y 139.812,Z 370.671,A -85,B 0,C 180,E1 -24906.285,E2 -24906.285} C_VEL
LIN {X 0,Y 137.21,Z 378.851,A -85,B 0,C 180,E1 -24910.55,E2 -24910.55} C_VEL
LIN {X 0,Y 135.319,Z 385.395,A -85,B 0,C 180,E1 -24914.946,E2 -24914.946} C_VEL
LIN {X 0,Y 134.131,Z 390.556,A -85,B 0,C 180,E1 -24919.43,E2 -24919.43} C_VEL
LIN {X 0,Y 133.545,Z 394.527,A -85,B 0,C 180,E1 -24923.955,E2 -24923.955} C_VEL
LIN {X 0,Y 133.4,Z 396.55,A -85,B 0,C 180,E1 -24926.977,E2 -24926.977} C_VEL
LIN {X 0,Y 133.477,Z 398.146,A -85,B 0,C 180,E1 -24929.997,E2 -24929.997} C_VEL
LIN {X 0,Y 133.405,Z 399.314,A -85,B 0,C 180,E1 -24933.017,E2 -24933.017} C_VEL
LIN {X 0,Y 133.57,Z 400.048,A -85,B 0,C 180,E1 -24936.037,E2 -24936.037} C_VEL
LIN {X 0,Y 134.625,Z 400.35,A -85,B 0,C 180,E1 -24942.05,E2 -24942.05} C_VEL
LIN {X 0,Y 136.945,Z 399.158,A -85,B 0,C 180,E1 -24947.93,E2 -24947.93} C_VEL
LIN {X 0,Y 139.248,Z 397.421,A -85,B 0,C 180,E1 -24951.721,E2 -24951.721} C_VEL
LIN {X 0,Y 140.38,Z 396.145,A -85,B 0,C 180,E1 -24954.042,E2 -24954.042} C_VEL
LIN {X 0,Y 140.98,Z 393.628,A -85,B 0,C 180,E1 -24957.962,E2 -24957.962} C_VEL
LIN {X 0,Y 142.135,Z 390.578,A -85,B 0,C 180,E1 -24961.761,E2 -24961.761} C_VEL
LIN {X 0,Y 144.061,Z 388.288,A -85,B 0,C 180,E1 -24963.805,E2 -24963.805} C_VEL
LIN {X 0,Y 149.862,Z 382.492,A -85,B 0,C 180,E1 -24967.56,E2 -24967.56} C_VEL
LIN {X 0,Y 155.946,Z 375.675,A -85,B 0,C 180,E1 -24970.799,E2 -24970.799} C_VEL
LIN {X 0,Y 161.417,Z 368.786,A -85,B 0,C 180,E1 -24973.29,E2 -24973.29} C_VEL
LIN {X 0,Y 167.126,Z 360.593,A -85,B 0,C 180,E1 -24975.629,E2 -24975.629} C_VEL
LIN {X 0,Y 173.162,Z 350.582,A -85,B 0,C 180,E1 -24977.786,E2 -24977.786} C_VEL
LIN {X 0,Y 178.258,Z 340.763,A -85,B 0,C 180,E1 -24979.367,E2 -24979.367} C_VEL
LIN {X 0,Y 183.42,Z 328.573,A -85,B 0,C 180,E1 -24980.883,E2 -24980.883} C_VEL
LIN {X 0,Y 187.459,Z 316.599,A -85,B 0,C 180,E1 -24981.93,E2 -24981.93} C_VEL
LIN {X 0,Y 190.569,Z 304.042,A -85,B 0,C 180,E1 -24982.722,E2 -24982.722} C_VEL
LIN {X 0,Y 192.733,Z 291.121,A -85,B 0,C 180,E1 -24983.238,E2 -24983.238} C_VEL
LIN {X 0,Y 194.439,Z 275.291,A -85,B 0,C 180,E1 -24983.809,E2 -24983.809} C_VEL
LIN {X 0,Y 191.957,Z 268.071,A -85,B 0,C 180,E1 -24986.607,E2 -24986.607} C_VEL
LIN {X 0,Y 189.61,Z 262.108,A -85,B 0,C 180,E1 -24989.735,E2 -24989.735} C_VEL
LIN {X 0,Y 188.251,Z 259.042,A -85,B 0,C 180,E1 -24991.925,E2 -24991.925} C_VEL
LIN {X 0,Y 186.778,Z 255.462,A -85,B 0,C 180,E1 -24995.21,E2 -24995.21} C_VEL
LIN {X 0,Y 185.831,Z 253.825,A -85,B 0,C 180,E1 -24998.274,E2 -24998.274} C_VEL
LIN {X 0,Y 185.365,Z 253.3,A -85,B 0,C 180,E1 -25002.342,E2 -25002.342} C_VEL
LIN {X 0,Y 186.068,Z 253.908,A -85,B 0,C 180,E1 -25006.9,E2 -25006.9} C_VEL
LIN {X 0,Y 186.76,Z 254.37,A -85,B 0,C 180,E1 -25008.711,E2 -25008.711} C_VEL
LIN {X 0,Y 188.28,Z 257.632,A -85,B 0,C 180,E1 -25012.128,E2 -25012.128} C_VEL
LIN {X 0,Y 189.263,Z 258.915,A -85,B 0,C 180,E1 -25013.603,E2 -25013.603} C_VEL
LIN {X 0,Y 190.722,Z 262.383,A -85,B 0,C 180,E1 -25015.773,E2 -25015.773} C_VEL
LIN {X 0,Y 192.739,Z 266.972,A -85,B 0,C 180,E1 -25018.188,E2 -25018.188} C_VEL
LIN {X 0,Y 194.711,Z 272.451,A -85,B 0,C 180,E1 -25020.352,E2 -25020.352} C_VEL
LIN {X 0,Y 191.983,Z 295.397,A -85,B 0,C 180,E1 -25021.186,E2 -25021.186} C_VEL
LIN {X 0,Y 189.125,Z 309.016,A -85,B 0,C 180,E1 -25021.899,E2 -25021.899} C_VEL
LIN {X 0,Y 185.517,Z 321.39,A -85,B 0,C 180,E1 -25022.932,E2 -25022.932} C_VEL
LIN {X 0,Y 180.847,Z 333.584,A -85,B 0,C 180,E1 -25024.309,E2 -25024.309} C_VEL
LIN {X 0,Y 175.389,Z 345.022,A -85,B 0,C 180,E1 -25026.04,E2 -25026.04} C_VEL
LIN {X 0,Y 169.542,Z 355.177,A -85,B 0,C 180,E1 -25028.111,E2 -25028.111} C_VEL
LIN {X 0,Y 162.763,Z 365.147,A -85,B 0,C 180,E1 -25030.806,E2 -25030.806} C_VEL
LIN {X 0,Y 157.024,Z 372.442,A -85,B 0,C 180,E1 -25033.438,E2 -25033.438} C_VEL
LIN {X 0,Y 150.958,Z 379.253,A -85,B 0,C 180,E1 -25036.671,E2 -25036.671} C_VEL
LIN {X 0,Y 144.937,Z 385.244,A -85,B 0,C 180,E1 -25040.607,E2 -25040.607} C_VEL
LIN {X 0,Y 139.486,Z 389.931,A -85,B 0,C 180,E1 -25044.925,E2 -25044.925} C_VEL
LIN {X 0,Y 135.885,Z 392.64,A -85,B 0,C 180,E1 -25048.457,E2 -25048.457} C_VEL
LIN {X 0,Y 132.852,Z 394.649,A -85,B 0,C 180,E1 -25052.184,E2 -25052.184} C_VEL
LIN {X 0,Y 130.141,Z 396.042,A -85,B 0,C 180,E1 -25056.442,E2 -25056.442} C_VEL
LIN {X 0,Y 127.964,Z 396.665,A -85,B 0,C 180,E1 -25061.226,E2 -25061.226} C_VEL
LIN {X 0,Y 126.508,Z 396.338,A -85,B 0,C 180,E1 -25066.234,E2 -25066.234} C_VEL
LIN {X 0,Y 125.763,Z 394.746,A -85,B 0,C 180,E1 -25072.074,E2 -25072.074} C_VEL
LIN {X 0,Y 125.845,Z 392.402,A -85,B 0,C 180,E1 -25076.895,E2 -25076.895} C_VEL
LIN {X 0,Y 126.454,Z 389.318,A -85,B 0,C 180,E1 -25081.377,E2 -25081.377} C_VEL
LIN {X 0,Y 127.381,Z 385.555,A -85,B 0,C 180,E1 -25085.56,E2 -25085.56} C_VEL
LIN {X 0,Y 128.689,Z 380.718,A -85,B 0,C 180,E1 -25089.795,E2 -25089.795} C_VEL
LIN {X 0,Y 131.045,Z 373.215,A -85,B 0,C 180,E1 -25094.867,E2 -25094.867} C_VEL
LIN {X 0,Y 133.934,Z 364.413,A -85,B 0,C 180,E1 -25099.422,E2 -25099.422} C_VEL
LIN {X 0,Y 137,Z 355.389,A -85,B 0,C 180,E1 -25103.005,E2 -25103.005} C_VEL
LIN {X 0,Y 140.265,Z 344.924,A -85,B 0,C 180,E1 -25106.258,E2 -25106.258} C_VEL
LIN {X 0,Y 143.38,Z 333.662,A -85,B 0,C 180,E1 -25108.95,E2 -25108.95} C_VEL
LIN {X 0,Y 146.407,Z 320.877,A -85,B 0,C 180,E1 -25111.223,E2 -25111.223} C_VEL
LIN {X 0,Y 148.61,Z 308.62,A -85,B 0,C 180,E1 -25112.837,E2 -25112.837} C_VEL
LIN {X 0,Y 150.486,Z 294.953,A -85,B 0,C 180,E1 -25114.022,E2 -25114.022} C_VEL
LIN {X 0,Y 152.35,Z 271.513,A -85,B 0,C 180,E1 -25115.206,E2 -25115.206} C_VEL
LIN {X 0,Y 154.207,Z 244.102,A -85,B 0,C 180,E1 -25116.501,E2 -25116.501} C_VEL
LIN {X 0,Y 147.868,Z 226.127,A -85,B 0,C 180,E1 -25119.286,E2 -25119.286} C_VEL
LIN {X 0,Y 138.621,Z 209.374,A -85,B 0,C 180,E1 -25123.211,E2 -25123.211} C_VEL
LIN {X 0,Y 133.764,Z 201.907,A -85,B 0,C 180,E1 -25125.452,E2 -25125.452} C_VEL
LIN {X 0,Y 131.377,Z 198.199,A -85,B 0,C 180,E1 -25126.624,E2 -25126.624} C_VEL
LIN {X 0,Y 129.643,Z 195.684,A -85,B 0,C 180,E1 -25127.522,E2 -25127.522} C_VEL
LIN {X 0,Y 129.22,Z 194.237,A -85,B 0,C 180,E1 -25128.151,E2 -25128.151} C_VEL
LIN {X 0,Y 129.133,Z 193.889,A -85,B 0,C 180,E1 -25129.063,E2 -25129.063} C_VEL
LIN {X 0,Y 129.108,Z 193.904,A -85,B 0,C 180,E1 -25132.402,E2 -25132.402} C_VEL
LIN {X 0,Y 129.028,Z 193.879,A -85,B 0,C 180,E1 -25135.836,E2 -25135.836} C_VEL
LIN {X 0,Y 129.017,Z 193.9,A -85,B 0,C 180,E1 -25139.361,E2 -25139.361} C_VEL
LIN {X 0,Y 128.959,Z 193.877,A -85,B 0,C 180,E1 -25145.17,E2 -25145.17} C_VEL
LIN {X 0,Y 128.945,Z 193.919,A -85,B 0,C 180,E1 -25150.851,E2 -25150.851} C_VEL
LIN {X 0,Y 128.919,Z 193.891,A -85,B 0,C 180,E1 -25155.133,E2 -25155.133} C_VEL
LIN {X 0,Y 128.941,Z 193.866,A -85,B 0,C 180,E1 -25159.74,E2 -25159.74} C_VEL
LIN {X 0,Y 128.961,Z 193.92,A -85,B 0,C 180,E1 -25164.835,E2 -25164.835} C_VEL
LIN {X 0,Y 129.02,Z 193.902,A -85,B 0,C 180,E1 -25170.645,E2 -25170.645} C_VEL
LIN {X 0,Y 129.112,Z 193.884,A -85,B 0,C 180,E1 -25177.604,E2 -25177.604} C_VEL
LIN {X 0,Y 129.154,Z 193.895,A -85,B 0,C 180,E1 -25180.945,E2 -25180.945} C_VEL
LIN {X 0,Y 129.394,Z 193.864,A -85,B 0,C 180,E1 -25187.88,E2 -25187.88} C_VEL
LIN {X 0,Y 129.468,Z 193.846,A -85,B 0,C 180,E1 -25190.629,E2 -25190.629} C_VEL
LIN {X 0,Y 130.072,Z 193.746,A -85,B 0,C 180,E1 -25200.001,E2 -25200.001} C_VEL
LIN {X 0,Y 129.475,Z 193.856,A -85,B 0,C 180,E1 -25209.373,E2 -25209.373} C_VEL
LIN {X 0,Y 129.304,Z 193.856,A -85,B 0,C 180,E1 -25212.558,E2 -25212.558} C_VEL
LIN {X 0,Y 129.088,Z 193.881,A -85,B 0,C 180,E1 -25219.068,E2 -25219.068} C_VEL
LIN {X 0,Y 129.039,Z 193.905,A -85,B 0,C 180,E1 -25222.412,E2 -25222.412} C_VEL
LIN {X 0,Y 129.005,Z 193.908,A -85,B 0,C 180,E1 -25229.362,E2 -25229.362} C_VEL
LIN {X 0,Y 129.007,Z 194.026,A -85,B 0,C 180,E1 -25235.194,E2 -25235.194} C_VEL
LIN {X 0,Y 129.181,Z 194.869,A -85,B 0,C 180,E1 -25235.922,E2 -25235.922} C_VEL
LIN {X 0,Y 130.876,Z 197.927,A -85,B 0,C 180,E1 -25236.926,E2 -25236.926} C_VEL
LIN {X 0,Y 132.044,Z 199.633,A -85,B 0,C 180,E1 -25237.502,E2 -25237.502} C_VEL
LIN {X 0,Y 137.144,Z 207.777,A -85,B 0,C 180,E1 -25239.96,E2 -25239.96} C_VEL
LIN {X 0,Y 142.46,Z 217.314,A -85,B 0,C 180,E1 -25242.353,E2 -25242.353} C_VEL
LIN {X 0,Y 149.109,Z 233.789,A -85,B 0,C 180,E1 -25245.329,E2 -25245.329} C_VEL
LIN {X 0,Y 154.05,Z 248.348,A -85,B 0,C 180,E1 -25247.503,E2 -25247.503} C_VEL
LIN {X 0,Y 150.624,Z 297.195,A -85,B 0,C 180,E1 -25249.87,E2 -25249.87} C_VEL
LIN {X 0,Y 148.694,Z 311.167,A -85,B 0,C 180,E1 -25251.005,E2 -25251.005} C_VEL
LIN {X 0,Y 146.493,Z 323.332,A -85,B 0,C 180,E1 -25252.503,E2 -25252.503} C_VEL
LIN {X 0,Y 143.726,Z 335.14,A -85,B 0,C 180,E1 -25254.499,E2 -25254.499} C_VEL
LIN {X 0,Y 141.006,Z 345.288,A -85,B 0,C 180,E1 -25256.749,E2 -25256.749} C_VEL
LIN {X 0,Y 137.754,Z 356.061,A -85,B 0,C 180,E1 -25259.818,E2 -25259.818} C_VEL
LIN {X 0,Y 134.912,Z 364.517,A -85,B 0,C 180,E1 -25262.88,E2 -25262.88} C_VEL
LIN {X 0,Y 132.292,Z 372.507,A -85,B 0,C 180,E1 -25266.516,E2 -25266.516} C_VEL
LIN {X 0,Y 129.709,Z 380.26,A -85,B 0,C 180,E1 -25271.025,E2 -25271.025} C_VEL
LIN {X 0,Y 127.932,Z 386.478,A -85,B 0,C 180,E1 -25275.684,E2 -25275.684} C_VEL
LIN {X 0,Y 126.861,Z 391.379,A -85,B 0,C 180,E1 -25280.43,E2 -25280.43} C_VEL
LIN {X 0,Y 126.373,Z 395.104,A -85,B 0,C 180,E1 -25285.212,E2 -25285.212} C_VEL
LIN {X 0,Y 126.392,Z 397.768,A -85,B 0,C 180,E1 -25289.997,E2 -25289.997} C_VEL
LIN {X 0,Y 126.33,Z 398.993,A -85,B 0,C 180,E1 -25293.186,E2 -25293.186} C_VEL
LIN {X 0,Y 126.521,Z 399.828,A -85,B 0,C 180,E1 -25296.375,E2 -25296.375} C_VEL
LIN {X 0,Y 127.674,Z 400.269,A -85,B 0,C 180,E1 -25302.716,E2 -25302.716} C_VEL
LIN {X 0,Y 130.175,Z 399.212,A -85,B 0,C 180,E1 -25308.897,E2 -25308.897} C_VEL
LIN {X 0,Y 132.504,Z 397.726,A -85,B 0,C 180,E1 -25312.636,E2 -25312.636} C_VEL
LIN {X 0,Y 136.85,Z 394.675,A -85,B 0,C 180,E1 -25317.525,E2 -25317.525} C_VEL
LIN {X 0,Y 141.298,Z 390.996,A -85,B 0,C 180,E1 -25321.48,E2 -25321.48} C_VEL
LIN {X 0,Y 144.061,Z 388.288,A -85,B 0,C 180,E1 -25323.805,E2 -25323.805} C_VEL
LIN {X 0,Y 146.154,Z 385.816,A -85,B 0,C 180,E1 -25325.762,E2 -25325.762} C_VEL
LIN {X 0,Y 148.404,Z 381.579,A -85,B 0,C 180,E1 -25329.147,E2 -25329.147} C_VEL
LIN {X 0,Y 150.992,Z 376.784,A -85,B 0,C 180,E1 -25332.307,E2 -25332.307} C_VEL
LIN {X 0,Y 153.506,Z 373.424,A -85,B 0,C 180,E1 -25333.867,E2 -25333.867} C_VEL
LIN {X 0,Y 159.913,Z 365.423,A -85,B 0,C 180,E1 -25336.477,E2 -25336.477} C_VEL
LIN {X 0,Y 166.083,Z 356.533,A -85,B 0,C 180,E1 -25338.682,E2 -25338.682} C_VEL
LIN {X 0,Y 171.793,Z 346.831,A -85,B 0,C 180,E1 -25340.544,E2 -25340.544} C_VEL
LIN {X 0,Y 177.801,Z 334.692,A -85,B 0,C 180,E1 -25342.231,E2 -25342.231} C_VEL
LIN {X 0,Y 182.569,Z 322.679,A -85,B 0,C 180,E1 -25343.469,E2 -25343.469} C_VEL
LIN {X 0,Y 186.56,Z 309.311,A -85,B 0,C 180,E1 -25344.432,E2 -25344.432} C_VEL
LIN {X 0,Y 189.324,Z 296.335,A -85,B 0,C 180,E1 -25345.019,E2 -25345.019} C_VEL
LIN {X 0,Y 191.444,Z 278.754,A -85,B 0,C 180,E1 -25345.664,E2 -25345.664} C_VEL
LIN {X 0,Y 189.334,Z 272.363,A -85,B 0,C 180,E1 -25348.376,E2 -25348.376} C_VEL
LIN {X 0,Y 187.682,Z 267.841,A -85,B 0,C 180,E1 -25350.965,E2 -25350.965} C_VEL
LIN {X 0,Y 186.659,Z 265.405,A -85,B 0,C 180,E1 -25352.802,E2 -25352.802} C_VEL
LIN {X 0,Y 185.518,Z 262.271,A -85,B 0,C 180,E1 -25355.73,E2 -25355.73} C_VEL
LIN {X 0,Y 184.717,Z 260.792,A -85,B 0,C 180,E1 -25358.636,E2 -25358.636} C_VEL
LIN {X 0,Y 184.333,Z 260.327,A -85,B 0,C 180,E1 -25362.385,E2 -25362.385} C_VEL
LIN {X 0,Y 185.01,Z 260.923,A -85,B 0,C 180,E1 -25366.824,E2 -25366.824} C_VEL
LIN {X 0,Y 185.566,Z 261.423,A -85,B 0,C 180,E1 -25368.393,E2 -25368.393} C_VEL
LIN {X 0,Y 187.264,Z 264.836,A -85,B 0,C 180,E1 -25372.219,E2 -25372.219} C_VEL
LIN {X 0,Y 188.104,Z 266.363,A -85,B 0,C 180,E1 -25373.563,E2 -25373.563} C_VEL
LIN {X 0,Y 190.578,Z 272.711,A -85,B 0,C 180,E1 -25377.119,E2 -25377.119} C_VEL
LIN {X 0,Y 191.719,Z 276.141,A -85,B 0,C 180,E1 -25378.518,E2 -25378.518} C_VEL
LIN {X 0,Y 189.111,Z 296.51,A -85,B 0,C 180,E1 -25379.25,E2 -25379.25} C_VEL
LIN {X 0,Y 186.203,Z 309.624,A -85,B 0,C 180,E1 -25379.935,E2 -25379.935} C_VEL
LIN {X 0,Y 182.739,Z 321.061,A -85,B 0,C 180,E1 -25380.877,E2 -25380.877} C_VEL
LIN {X 0,Y 178.35,Z 332.217,A -85,B 0,C 180,E1 -25382.067,E2 -25382.067} C_VEL
LIN {X 0,Y 172.547,Z 344.117,A -85,B 0,C 180,E1 -25383.778,E2 -25383.778} C_VEL
LIN {X 0,Y 166.845,Z 353.916,A -85,B 0,C 180,E1 -25385.678,E2 -25385.678} C_VEL
LIN {X 0,Y 161.227,Z 362.1,A -85,B 0,C 180,E1 -25387.698,E2 -25387.698} C_VEL
LIN {X 0,Y 154.502,Z 370.586,A -85,B 0,C 180,E1 -25390.482,E2 -25390.482} C_VEL
LIN {X 0,Y 147.667,Z 378.023,A -85,B 0,C 180,E1 -25393.765,E2 -25393.765} C_VEL
LIN {X 0,Y 141.632,Z 383.835,A -85,B 0,C 180,E1 -25397.32,E2 -25397.32} C_VEL
LIN {X 0,Y 135.881,Z 388.702,A -85,B 0,C 180,E1 -25401.421,E2 -25401.421} C_VEL
LIN {X 0,Y 131.273,Z 392.013,A -85,B 0,C 180,E1 -25405.358,E2 -25405.358} C_VEL
LIN {X 0,Y 127.189,Z 394.532,A -85,B 0,C 180,E1 -25409.82,E2 -25409.82} C_VEL
LIN {X 0,Y 123.896,Z 396.108,A -85,B 0,C 180,E1 -25414.557,E2 -25414.557} C_VEL
LIN {X 0,Y 120.889,Z 396.822,A -85,B 0,C 180,E1 -25420.914,E2 -25420.914} C_VEL
LIN {X 0,Y 119.606,Z 396.447,A -85,B 0,C 180,E1 -25425.167,E2 -25425.167} C_VEL
LIN {X 0,Y 118.79,Z 395.21,A -85,B 0,C 180,E1 -25430.273,E2 -25430.273} C_VEL
LIN {X 0,Y 118.697,Z 392.741,A -85,B 0,C 180,E1 -25435.987,E2 -25435.987} C_VEL
LIN {X 0,Y 119.437,Z 388.832,A -85,B 0,C 180,E1 -25441.959,E2 -25441.959} C_VEL
LIN {X 0,Y 120.689,Z 384.056,A -85,B 0,C 180,E1 -25447.222,E2 -25447.222} C_VEL
LIN {X 0,Y 122.547,Z 377.733,A -85,B 0,C 180,E1 -25452.481,E2 -25452.481} C_VEL
LIN {X 0,Y 124.983,Z 370.701,A -85,B 0,C 180,E1 -25457.005,E2 -25457.005} C_VEL
LIN {X 0,Y 128.174,Z 361.593,A -85,B 0,C 180,E1 -25461.56,E2 -25461.56} C_VEL
LIN {X 0,Y 131.616,Z 351.475,A -85,B 0,C 180,E1 -25465.409,E2 -25465.409} C_VEL
LIN {X 0,Y 135.005,Z 340.827,A -85,B 0,C 180,E1 -25468.512,E2 -25468.512} C_VEL
LIN {X 0,Y 138.139,Z 329.311,A -85,B 0,C 180,E1 -25471.096,E2 -25471.096} C_VEL
LIN {X 0,Y 140.755,Z 317.69,A -85,B 0,C 180,E1 -25473.046,E2 -25473.046} C_VEL
LIN {X 0,Y 143.1,Z 304.303,A -85,B 0,C 180,E1 -25474.669,E2 -25474.669} C_VEL
LIN {X 0,Y 144.786,Z 291.594,A -85,B 0,C 180,E1 -25475.648,E2 -25475.648} C_VEL
LIN {X 0,Y 148.124,Z 245.431,A -85,B 0,C 180,E1 -25477.931,E2 -25477.931} C_VEL
LIN {X 0,Y 142.527,Z 229.683,A -85,B 0,C 180,E1 -25480.523,E2 -25480.523} C_VEL
LIN {X 0,Y 133.801,Z 213.66,A -85,B 0,C 180,E1 -25484.507,E2 -25484.507} C_VEL
LIN {X 0,Y 126.936,Z 203.034,A -85,B 0,C 180,E1 -25487.95,E2 -25487.95} C_VEL
LIN {X 0,Y 124.561,Z 199.335,A -85,B 0,C 180,E1 -25489.279,E2 -25489.279} C_VEL
LIN {X 0,Y 122.722,Z 197.049,A -85,B 0,C 180,E1 -25490.312,E2 -25490.312} C_VEL
LIN {X 0,Y 122.101,Z 195.256,A -85,B 0,C 180,E1 -25491.062,E2 -25491.062} C_VEL
LIN {X 0,Y 122.047,Z 194.833,A -85,B 0,C 180,E1 -25491.742,E2 -25491.742} C_VEL
LIN {X 0,Y 121.941,Z 194.762,A -85,B 0,C 180,E1 -25497.46,E2 -25497.46} C_VEL
LIN {X 0,Y 121.9,Z 194.802,A -85,B 0,C 180,E1 -25501.261,E2 -25501.261} C_VEL
LIN {X 0,Y 121.884,Z 194.754,A -85,B 0,C 180,E1 -25506.174,E2 -25506.174} C_VEL
LIN {X 0,Y 121.881,Z 194.803,A -85,B 0,C 180,E1 -25511.445,E2 -25511.445} C_VEL
LIN {X 0,Y 121.869,Z 194.741,A -85,B 0,C 180,E1 -25518.568,E2 -25518.568} C_VEL
LIN {X 0,Y 121.913,Z 194.798,A -85,B 0,C 180,E1 -25524.799,E2 -25524.799} C_VEL
LIN {X 0,Y 121.93,Z 194.78,A -85,B 0,C 180,E1 -25529.842,E2 -25529.842} C_VEL
LIN {X 0,Y 121.985,Z 194.771,A -85,B 0,C 180,E1 -25536.217,E2 -25536.217} C_VEL
LIN {X 0,Y 122.048,Z 194.778,A -85,B 0,C 180,E1 -25539.789,E2 -25539.789} C_VEL
LIN {X 0,Y 122.243,Z 194.747,A -85,B 0,C 180,E1 -25546.706,E2 -25546.706} C_VEL
LIN {X 0,Y 122.406,Z 194.73,A -85,B 0,C 180,E1 -25550.083,E2 -25550.083} C_VEL
LIN {X 0,Y 122.564,Z 194.717,A -85,B 0,C 180,E1 -25556.714,E2 -25556.714} C_VEL
LIN {X 0,Y 123.025,Z 194.62,A -85,B 0,C 180,E1 -25560.001,E2 -25560.001} C_VEL
LIN {X 0,Y 122.413,Z 194.696,A -85,B 0,C 180,E1 -25566.595,E2 -25566.595} C_VEL
LIN {X 0,Y 122.401,Z 194.739,A -85,B 0,C 180,E1 -25569.92,E2 -25569.92} C_VEL
LIN {X 0,Y 122.193,Z 194.729,A -85,B 0,C 180,E1 -25573.302,E2 -25573.302} C_VEL
LIN {X 0,Y 121.993,Z 194.781,A -85,B 0,C 180,E1 -25580.224,E2 -25580.224} C_VEL
LIN {X 0,Y 121.916,Z 194.772,A -85,B 0,C 180,E1 -25583.8,E2 -25583.8} C_VEL
LIN {X 0,Y 121.921,Z 194.8,A -85,B 0,C 180,E1 -25590.151,E2 -25590.151} C_VEL
LIN {X 0,Y 121.96,Z 195.057,A -85,B 0,C 180,E1 -25592.457,E2 -25592.457} C_VEL
LIN {X 0,Y 122.235,Z 196.112,A -85,B 0,C 180,E1 -25593.109,E2 -25593.109} C_VEL
LIN {X 0,Y 123.934,Z 198.839,A -85,B 0,C 180,E1 -25594.179,E2 -25594.179} C_VEL
LIN {X 0,Y 124.971,Z 200.203,A -85,B 0,C 180,E1 -25594.752,E2 -25594.752} C_VEL
LIN {X 0,Y 132.197,Z 211.676,A -85,B 0,C 180,E1 -25598.537,E2 -25598.537} C_VEL
LIN {X 0,Y 137.547,Z 221.504,A -85,B 0,C 180,E1 -25601.138,E2 -25601.138} C_VEL
LIN {X 0,Y 143.929,Z 237.809,A -85,B 0,C 180,E1 -25604.216,E2 -25604.216} C_VEL
LIN {X 0,Y 148.004,Z 250.022,A -85,B 0,C 180,E1 -25606.122,E2 -25606.122} C_VEL
LIN {X 0,Y 144.486,Z 297.418,A -85,B 0,C 180,E1 -25608.488,E2 -25608.488} C_VEL
LIN {X 0,Y 142.49,Z 311.284,A -85,B 0,C 180,E1 -25609.654,E2 -25609.654} C_VEL
LIN {X 0,Y 140.212,Z 323.389,A -85,B 0,C 180,E1 -25611.201,E2 -25611.201} C_VEL
LIN {X 0,Y 137.075,Z 335.914,A -85,B 0,C 180,E1 -25613.411,E2 -25613.411} C_VEL
LIN {X 0,Y 133.875,Z 347.196,A -85,B 0,C 180,E1 -25616.094,E2 -25616.094} C_VEL
LIN {X 0,Y 130.643,Z 357.39,A -85,B 0,C 180,E1 -25619.264,E2 -25619.264} C_VEL
LIN {X 0,Y 128.003,Z 364.895,A -85,B 0,C 180,E1 -25622.177,E2 -25622.177} C_VEL
LIN {X 0,Y 124.807,Z 374.155,A -85,B 0,C 180,E1 -25626.782,E2 -25626.782} C_VEL
LIN {X 0,Y 122.216,Z 381.57,A -85,B 0,C 180,E1 -25631.559,E2 -25631.559} C_VEL
LIN {X 0,Y 120.551,Z 387.51,A -85,B 0,C 180,E1 -25636.511,E2 -25636.511} C_VEL
LIN {X 0,Y 119.602,Z 392.15,A -85,B 0,C 180,E1 -25641.549,E2 -25641.549} C_VEL
LIN {X 0,Y 119.248,Z 395.641,A -85,B 0,C 180,E1 -25646.618,E2 -25646.618} C_VEL
LIN {X 0,Y 119.322,Z 397.374,A -85,B 0,C 180,E1 -25649.996,E2 -25649.996} C_VEL
LIN {X 0,Y 119.26,Z 398.663,A -85,B 0,C 180,E1 -25653.375,E2 -25653.375} C_VEL
LIN {X 0,Y 119.461,Z 399.56,A -85,B 0,C 180,E1 -25656.754,E2 -25656.754} C_VEL
LIN {X 0,Y 119.948,Z 400.077,A -85,B 0,C 180,E1 -25660.12,E2 -25660.12} C_VEL
LIN {X 0,Y 121.921,Z 399.908,A -85,B 0,C 180,E1 -25666.747,E2 -25666.747} C_VEL
LIN {X 0,Y 125.395,Z 398.249,A -85,B 0,C 180,E1 -25673.095,E2 -25673.095} C_VEL
LIN {X 0,Y 127.787,Z 396.852,A -85,B 0,C 180,E1 -25676.099,E2 -25676.099} C_VEL
LIN {X 0,Y 132.141,Z 393.946,A -85,B 0,C 180,E1 -25680.345,E2 -25680.345} C_VEL
LIN {X 0,Y 137.679,Z 389.363,A -85,B 0,C 180,E1 -25685.032,E2 -25685.032} C_VEL
LIN {X 0,Y 144.348,Z 383.246,A -85,B 0,C 180,E1 -25689.263,E2 -25689.263} C_VEL
LIN {X 0,Y 150.703,Z 376.661,A -85,B 0,C 180,E1 -25692.543,E2 -25692.543} C_VEL
LIN {X 0,Y 153.506,Z 373.424,A -85,B 0,C 180,E1 -25693.867,E2 -25693.867} C_VEL
LIN {X 0,Y 155.077,Z 371.117,A -85,B 0,C 180,E1 -25694.928,E2 -25694.928} C_VEL
LIN {X 0,Y 157.83,Z 363.82,A -85,B 0,C 180,E1 -25698.967,E2 -25698.967} C_VEL
LIN {X 0,Y 159.478,Z 361.16,A -85,B 0,C 180,E1 -25699.858,E2 -25699.858} C_VEL
LIN {X 0,Y 166.14,Z 351.21,A -85,B 0,C 180,E1 -25701.981,E2 -25701.981} C_VEL
LIN {X 0,Y 172.292,Z 340.254,A -85,B 0,C 180,E1 -25703.665,E2 -25703.665} C_VEL
LIN {X 0,Y 177.863,Z 328.034,A -85,B 0,C 180,E1 -25705.07,E2 -25705.07} C_VEL
LIN {X 0,Y 181.825,Z 317.065,A -85,B 0,C 180,E1 -25705.979,E2 -25705.979} C_VEL
LIN {X 0,Y 185.194,Z 304.636,A -85,B 0,C 180,E1 -25706.715,E2 -25706.715} C_VEL
LIN {X 0,Y 187.664,Z 290.862,A -85,B 0,C 180,E1 -25707.254,E2 -25707.254} C_VEL
LIN {X 0,Y 188.656,Z 282.437,A -85,B 0,C 180,E1 -25707.548,E2 -25707.548} C_VEL
LIN {X 0,Y 187.16,Z 277.496,A -85,B 0,C 180,E1 -25709.863,E2 -25709.863} C_VEL
LIN {X 0,Y 185.841,Z 273.592,A -85,B 0,C 180,E1 -25712.22,E2 -25712.22} C_VEL
LIN {X 0,Y 184.961,Z 271.27,A -85,B 0,C 180,E1 -25714.189,E2 -25714.189} C_VEL
LIN {X 0,Y 184.281,Z 269.077,A -85,B 0,C 180,E1 -25716.24,E2 -25716.24} C_VEL
LIN {X 0,Y 183.603,Z 267.728,A -85,B 0,C 180,E1 -25719.064,E2 -25719.064} C_VEL
LIN {X 0,Y 183.366,Z 267.398,A -85,B 0,C 180,E1 -25723.363,E2 -25723.363} C_VEL
LIN {X 0,Y 184.363,Z 268.319,A -85,B 0,C 180,E1 -25727.984,E2 -25727.984} C_VEL
LIN {X 0,Y 186.072,Z 271.843,A -85,B 0,C 180,E1 -25732.034,E2 -25732.034} C_VEL
LIN {X 0,Y 187.122,Z 274.585,A -85,B 0,C 180,E1 -25733.874,E2 -25733.874} C_VEL
LIN {X 0,Y 188.659,Z 279.005,A -85,B 0,C 180,E1 -25736.253,E2 -25736.253} C_VEL
LIN {X 0,Y 188.938,Z 279.969,A -85,B 0,C 180,E1 -25736.658,E2 -25736.658} C_VEL
LIN {X 0,Y 186.447,Z 297.775,A -85,B 0,C 180,E1 -25737.269,E2 -25737.269} C_VEL
LIN {X 0,Y 183.61,Z 309.941,A -85,B 0,C 180,E1 -25737.894,E2 -25737.894} C_VEL
LIN {X 0,Y 179.677,Z 322.254,A -85,B 0,C 180,E1 -25738.885,E2 -25738.885} C_VEL
LIN {X 0,Y 175.325,Z 332.831,A -85,B 0,C 180,E1 -25739.999,E2 -25739.999} C_VEL
LIN {X 0,Y 169.605,Z 344.133,A -85,B 0,C 180,E1 -25741.584,E2 -25741.584} C_VEL
LIN {X 0,Y 163.572,Z 354.022,A -85,B 0,C 180,E1 -25743.441,E2 -25743.441} C_VEL
LIN {X 0,Y 157.089,Z 362.956,A -85,B 0,C 180,E1 -25745.644,E2 -25745.644} C_VEL
LIN {X 0,Y 149.309,Z 372.147,A -85,B 0,C 180,E1 -25748.733,E2 -25748.733} C_VEL
LIN {X 0,Y 141.977,Z 379.513,A -85,B 0,C 180,E1 -25752.156,E2 -25752.156} C_VEL
LIN {X 0,Y 134.958,Z 385.61,A -85,B 0,C 180,E1 -25756.24,E2 -25756.24} C_VEL
LIN {X 0,Y 128.122,Z 390.658,A -85,B 0,C 180,E1 -25761.18,E2 -25761.18} C_VEL
LIN {X 0,Y 123.971,Z 393.212,A -85,B 0,C 180,E1 -25764.91,E2 -25764.91} C_VEL
LIN {X 0,Y 120.387,Z 395.115,A -85,B 0,C 180,E1 -25768.884,E2 -25768.884} C_VEL
LIN {X 0,Y 117.426,Z 396.319,A -85,B 0,C 180,E1 -25773.088,E2 -25773.088} C_VEL
LIN {X 0,Y 114.969,Z 396.886,A -85,B 0,C 180,E1 -25777.681,E2 -25777.681} C_VEL
LIN {X 0,Y 112.972,Z 396.664,A -85,B 0,C 180,E1 -25783.179,E2 -25783.179} C_VEL
LIN {X 0,Y 111.813,Z 395.436,A -85,B 0,C 180,E1 -25788.958,E2 -25788.958} C_VEL
LIN {X 0,Y 111.563,Z 392.826,A -85,B 0,C 180,E1 -25795.467,E2 -25795.467} C_VEL
LIN {X 0,Y 112.206,Z 389.298,A -85,B 0,C 180,E1 -25801.265,E2 -25801.265} C_VEL
LIN {X 0,Y 113.27,Z 385.252,A -85,B 0,C 180,E1 -25806.197,E2 -25806.197} C_VEL
LIN {X 0,Y 114.824,Z 379.916,A -85,B 0,C 180,E1 -25811.26,E2 -25811.26} C_VEL
LIN {X 0,Y 117.082,Z 373.376,A -85,B 0,C 180,E1 -25816.111,E2 -25816.111} C_VEL
LIN {X 0,Y 120.118,Z 365.05,A -85,B 0,C 180,E1 -25820.915,E2 -25820.915} C_VEL
LIN {X 0,Y 123.633,Z 355.473,A -85,B 0,C 180,E1 -25825.112,E2 -25825.112} C_VEL
LIN {X 0,Y 127.313,Z 344.714,A -85,B 0,C 180,E1 -25828.728,E2 -25828.728} C_VEL
LIN {X 0,Y 130.633,Z 333.677,A -85,B 0,C 180,E1 -25831.545,E2 -25831.545} C_VEL
LIN {X 0,Y 133.841,Z 321.205,A -85,B 0,C 180,E1 -25833.916,E2 -25833.916} C_VEL
LIN {X 0,Y 136.192,Z 309.234,A -85,B 0,C 180,E1 -25835.608,E2 -25835.608} C_VEL
LIN {X 0,Y 138.254,Z 295.703,A -85,B 0,C 180,E1 -25836.865,E2 -25836.865} C_VEL
LIN {X 0,Y 140.162,Z 274.344,A -85,B 0,C 180,E1 -25838.024,E2 -25838.024} C_VEL
LIN {X 0,Y 142.097,Z 247.058,A -85,B 0,C 180,E1 -25839.414,E2 -25839.414} C_VEL
LIN {X 0,Y 137.33,Z 233.389,A -85,B 0,C 180,E1 -25841.815,E2 -25841.815} C_VEL
LIN {X 0,Y 129.26,Z 218.318,A -85,B 0,C 180,E1 -25845.747,E2 -25845.747} C_VEL
LIN {X 0,Y 122.667,Z 207.904,A -85,B 0,C 180,E1 -25849.325,E2 -25849.325} C_VEL
LIN {X 0,Y 120.436,Z 204.509,A -85,B 0,C 180,E1 -25850.665,E2 -25850.665} C_VEL
LIN {X 0,Y 118.221,Z 201.15,A -85,B 0,C 180,E1 -25852.053,E2 -25852.053} C_VEL
LIN {X 0,Y 116.938,Z 199.691,A -85,B 0,C 180,E1 -25852.832,E2 -25852.832} C_VEL
LIN {X 0,Y 115.34,Z 197.318,A -85,B 0,C 180,E1 -25853.941,E2 -25853.941} C_VEL
LIN {X 0,Y 114.967,Z 196.035,A -85,B 0,C 180,E1 -25854.644,E2 -25854.644} C_VEL
LIN {X 0,Y 114.894,Z 195.714,A -85,B 0,C 180,E1 -25855.356,E2 -25855.356} C_VEL
LIN {X 0,Y 114.857,Z 195.68,A -85,B 0,C 180,E1 -25861.061,E2 -25861.061} C_VEL
LIN {X 0,Y 114.781,Z 195.642,A -85,B 0,C 180,E1 -25867.76,E2 -25867.76} C_VEL
LIN {X 0,Y 114.792,Z 195.683,A -85,B 0,C 180,E1 -25872.722,E2 -25872.722} C_VEL
LIN {X 0,Y 114.792,Z 195.621,A -85,B 0,C 180,E1 -25877.667,E2 -25877.667} C_VEL
LIN {X 0,Y 114.789,Z 195.661,A -85,B 0,C 180,E1 -25882.748,E2 -25882.748} C_VEL
LIN {X 0,Y 114.858,Z 195.659,A -85,B 0,C 180,E1 -25888.947,E2 -25888.947} C_VEL
LIN {X 0,Y 114.95,Z 195.646,A -85,B 0,C 180,E1 -25896.512,E2 -25896.512} C_VEL
LIN {X 0,Y 115.013,Z 195.65,A -85,B 0,C 180,E1 -25902.212,E2 -25902.212} C_VEL
LIN {X 0,Y 115.253,Z 195.622,A -85,B 0,C 180,E1 -25907.347,E2 -25907.347} C_VEL
LIN {X 0,Y 115.353,Z 195.597,A -85,B 0,C 180,E1 -25913.003,E2 -25913.003} C_VEL
LIN {X 0,Y 115.953,Z 195.497,A -85,B 0,C 180,E1 -25920.002,E2 -25920.002} C_VEL
LIN {X 0,Y 115.356,Z 195.578,A -85,B 0,C 180,E1 -25927,E2 -25927} C_VEL
LIN {X 0,Y 115.21,Z 195.606,A -85,B 0,C 180,E1 -25932.559,E2 -25932.559} C_VEL
LIN {X 0,Y 114.971,Z 195.619,A -85,B 0,C 180,E1 -25937.798,E2 -25937.798} C_VEL
LIN {X 0,Y 114.898,Z 195.648,A -85,B 0,C 180,E1 -25943.429,E2 -25943.429} C_VEL
LIN {X 0,Y 114.85,Z 195.863,A -85,B 0,C 180,E1 -25948.811,E2 -25948.811} C_VEL
LIN {X 0,Y 115.085,Z 196.8,A -85,B 0,C 180,E1 -25949.6,E2 -25949.6} C_VEL
LIN {X 0,Y 116.757,Z 199.687,A -85,B 0,C 180,E1 -25950.83,E2 -25950.83} C_VEL
LIN {X 0,Y 118.274,Z 201.31,A -85,B 0,C 180,E1 -25951.762,E2 -25951.762} C_VEL
LIN {X 0,Y 120.197,Z 204.331,A -85,B 0,C 180,E1 -25952.993,E2 -25952.993} C_VEL
LIN {X 0,Y 126.509,Z 214.419,A -85,B 0,C 180,E1 -25956.634,E2 -25956.634} C_VEL
LIN {X 0,Y 132.278,Z 224.744,A -85,B 0,C 180,E1 -25959.612,E2 -25959.612} C_VEL
LIN {X 0,Y 138.263,Z 240.248,A -85,B 0,C 180,E1 -25962.757,E2 -25962.757} C_VEL
LIN {X 0,Y 142.049,Z 251.707,A -85,B 0,C 180,E1 -25964.67,E2 -25964.67} C_VEL
LIN {X 0,Y 138.44,Z 297.128,A -85,B 0,C 180,E1 -25966.981,E2 -25966.981} C_VEL
